REGION Network 3: Stopper02
   "InstSq_Stopper02"(INIT_SQ := #tempInit,   // "Sq_Process_Stopper"
                      ACK_EF := #tempAck,
                      SW_AUTO := #tempSwAuto,
                      SW_TAP := #tempSwTap,
                      SW_MAN := #tempSwMan,
                      T_PUSH := #tempPush,
                      ixStart := "InstSq_Process_Lift1".qxReadyForNextWT,
                      ixCarrierPresent := "FG_TS_Stopper02_B_Detect",
                      ixCheckTargetReached := true,
                      ixTargetReached := "FG_TS_Lift01_B_Detect",
                      itStopperRelease := t#150ms,
                      signals := #station.signals,
                      sq := #station.stepSeqs.stepSeq[2],
                      cylinder_stopper := "TransportActors".Stopper02);
END_REGION

REGION Network 4: Lift 1
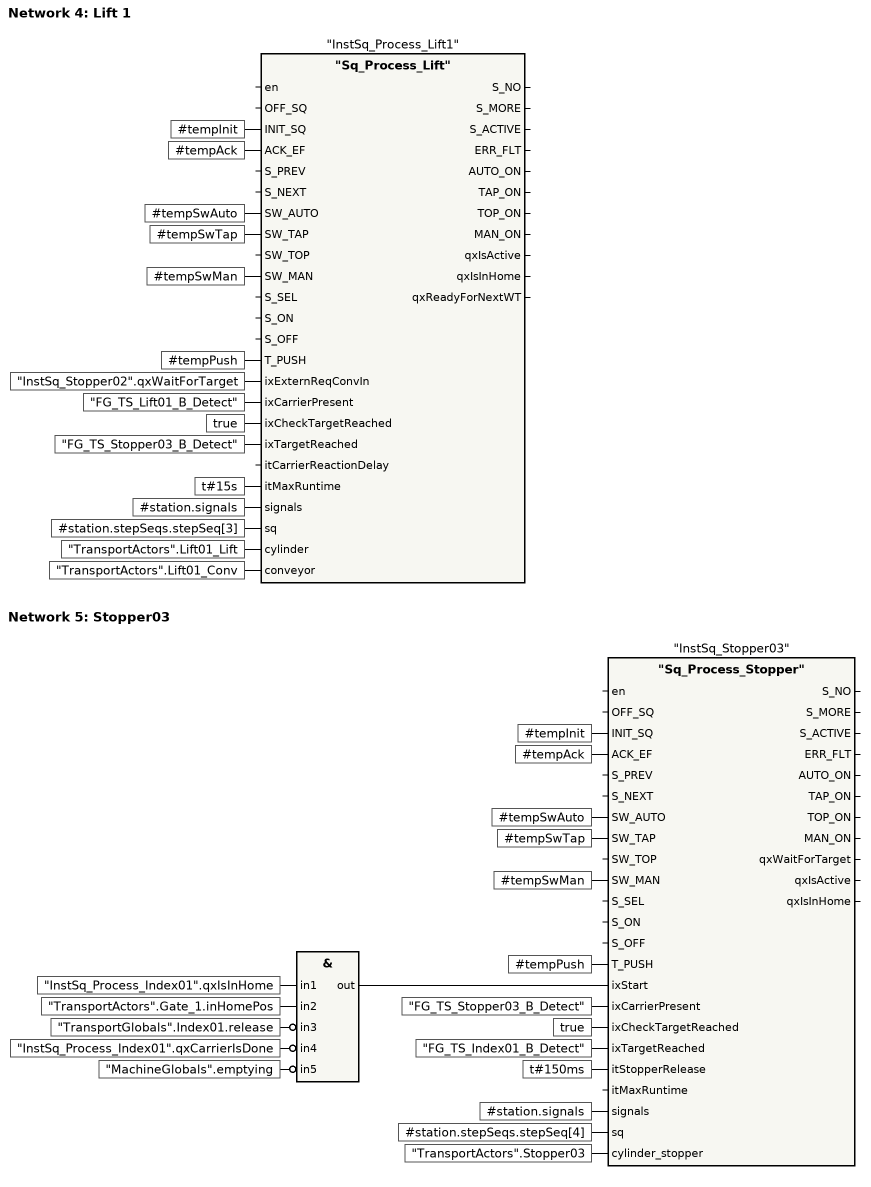
   "InstSq_Process_Lift1"(INIT_SQ := #tempInit,   // "Sq_Process_Lift"
                          ACK_EF := #tempAck,
                          SW_AUTO := #tempSwAuto,
                          SW_TAP := #tempSwTap,
                          SW_MAN := #tempSwMan,
                          T_PUSH := #tempPush,
                          ixExternReqConvIn := "InstSq_Stopper02".qxWaitForTarget,
                          ixCarrierPresent := "FG_TS_Lift01_B_Detect",
                          ixCheckTargetReached := true,
                          ixTargetReached := "FG_TS_Stopper03_B_Detect",
                          itMaxRuntime := t#15s,
                          signals := #station.signals,
                          sq := #station.stepSeqs.stepSeq[3],
                          cylinder := "TransportActors".Lift01_Lift,
                          conveyor := "TransportActors".Lift01_Conv);
END_REGION

REGION Network 5: Stopper03
   "InstSq_Stopper03"(INIT_SQ := #tempInit,   // "Sq_Process_Stopper"
                      ACK_EF := #tempAck,
                      SW_AUTO := #tempSwAuto,
                      SW_TAP := #tempSwTap,
                      SW_MAN := #tempSwMan,
                      T_PUSH := #tempPush,
                      ixStart := "InstSq_Process_Index01".qxIsInHome AND "TransportActors".Gate_1.inHomePos AND NOT "TransportGlobals".Index01.release AND NOT "InstSq_Process_Index01".qxCarrierIsDone AND NOT "MachineGlobals".emptying,
                      ixCarrierPresent := "FG_TS_Stopper03_B_Detect",
                      ixCheckTargetReached := true,
                      ixTargetReached := "FG_TS_Index01_B_Detect",
                      itStopperRelease := t#150ms,
                      signals := #station.signals,
                      sq := #station.stepSeqs.stepSeq[4],
                      cylinder_stopper := "TransportActors".Stopper03);
END_REGION

REGION Network 6: Index01
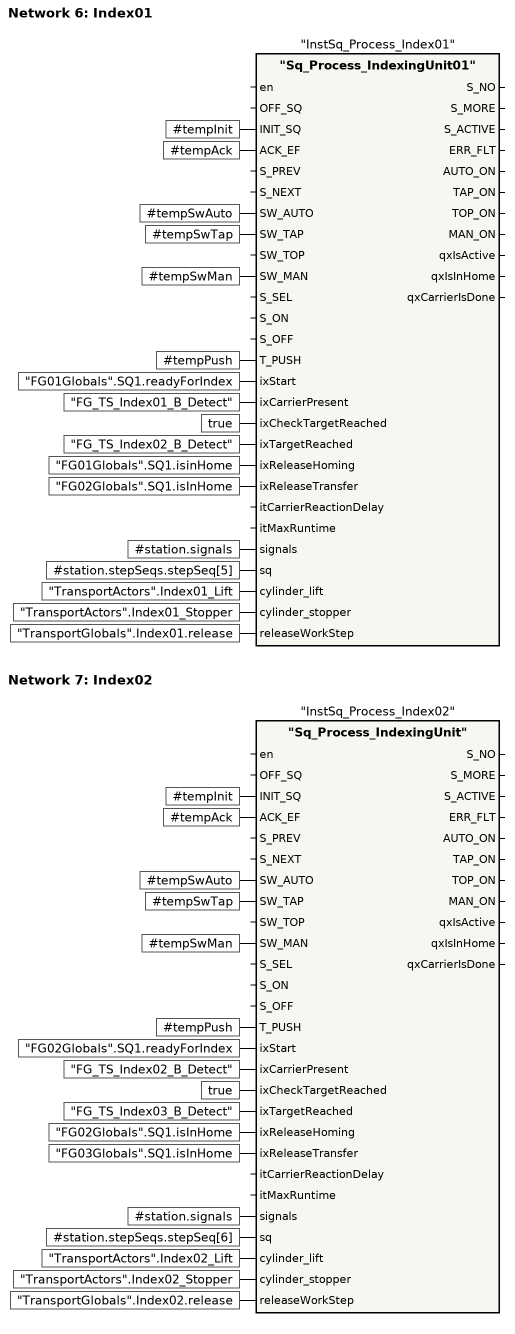
   "InstSq_Process_Index01"(INIT_SQ := #tempInit,   // "Sq_Process_IndexingUnit01"
                           ACK_EF := #tempAck,
                           SW_AUTO := #tempSwAuto,
                           SW_TAP := #tempSwTap,
                           SW_MAN := #tempSwMan,
                           T_PUSH := #tempPush,
                           ixStart := "FG01Globals".SQ1.readyForIndex,
                           ixCarrierPresent := "FG_TS_Index01_B_Detect",
                           ixCheckTargetReached := true,
                           ixTargetReached := "FG_TS_Index02_B_Detect",
                           ixReleaseHoming := "FG01Globals".SQ1.isinHome,
                           ixReleaseTransfer := "FG02Globals".SQ1.isInHome,
                           signals := #station.signals,
                           sq := #station.stepSeqs.stepSeq[5],
                           cylinder_lift := "TransportActors".Index01_Lift,
                           cylinder_stopper := "TransportActors".Index01_Stopper,
                           releaseWorkStep := "TransportGlobals".Index01.release);
END_REGION

REGION Network 7: Index02
   "InstSq_Process_Index02"(INIT_SQ := #tempInit,   // "Sq_Process_IndexingUnit"
                           ACK_EF := #tempAck,
                           SW_AUTO := #tempSwAuto,
                           SW_TAP := #tempSwTap,
                           SW_MAN := #tempSwMan,
                           T_PUSH := #tempPush,
                           ixStart := "FG02Globals".SQ1.readyForIndex,
                           ixCarrierPresent := "FG_TS_Index02_B_Detect",
                           ixCheckTargetReached := true,
                           ixTargetReached := "FG_TS_Index03_B_Detect",
                           ixReleaseHoming := "FG02Globals".SQ1.isInHome,
                           ixReleaseTransfer := "FG03Globals".SQ1.isInHome,
                           signals := #station.signals,
                           sq := #station.stepSeqs.stepSeq[6],
                           cylinder_lift := "TransportActors".Index02_Lift,
                           cylinder_stopper := "TransportActors".Index02_Stopper,
                           releaseWorkStep := "TransportGlobals".Index02.release);
END_REGION

REGION Network 8: Index03
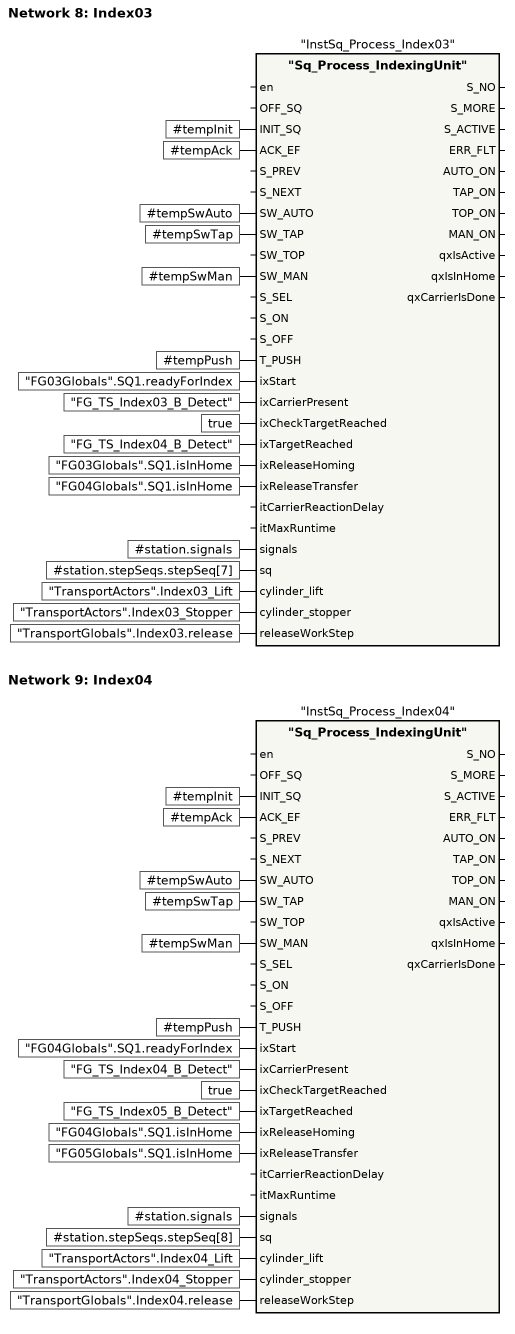
   "InstSq_Process_Index03"(INIT_SQ := #tempInit,   // "Sq_Process_IndexingUnit"
                           ACK_EF := #tempAck,
                           SW_AUTO := #tempSwAuto,
                           SW_TAP := #tempSwTap,
                           SW_MAN := #tempSwMan,
                           T_PUSH := #tempPush,
                           ixStart := "FG03Globals".SQ1.readyForIndex,
                           ixCarrierPresent := "FG_TS_Index03_B_Detect",
                           ixCheckTargetReached := true,
                           ixTargetReached := "FG_TS_Index04_B_Detect",
                           ixReleaseHoming := "FG03Globals".SQ1.isInHome,
                           ixReleaseTransfer := "FG04Globals".SQ1.isInHome,
                           signals := #station.signals,
                           sq := #station.stepSeqs.stepSeq[7],
                           cylinder_lift := "TransportActors".Index03_Lift,
                           cylinder_stopper := "TransportActors".Index03_Stopper,
                           releaseWorkStep := "TransportGlobals".Index03.release);
END_REGION

REGION Network 9: Index04
   "InstSq_Process_Index04"(INIT_SQ := #tempInit,   // "Sq_Process_IndexingUnit"
                           ACK_EF := #tempAck,
                           SW_AUTO := #tempSwAuto,
                           SW_TAP := #tempSwTap,
                           SW_MAN := #tempSwMan,
                           T_PUSH := #tempPush,
                           ixStart := "FG04Globals".SQ1.readyForIndex,
                           ixCarrierPresent := "FG_TS_Index04_B_Detect",
                           ixCheckTargetReached := true,
                           ixTargetReached := "FG_TS_Index05_B_Detect",
                           ixReleaseHoming := "FG04Globals".SQ1.isInHome,
                           ixReleaseTransfer := "FG05Globals".SQ1.isInHome,
                           signals := #station.signals,
                           sq := #station.stepSeqs.stepSeq[8],
                           cylinder_lift := "TransportActors".Index04_Lift,
                           cylinder_stopper := "TransportActors".Index04_Stopper,
                           releaseWorkStep := "TransportGlobals".Index04.release);
END_REGION

REGION Network 10: Index05
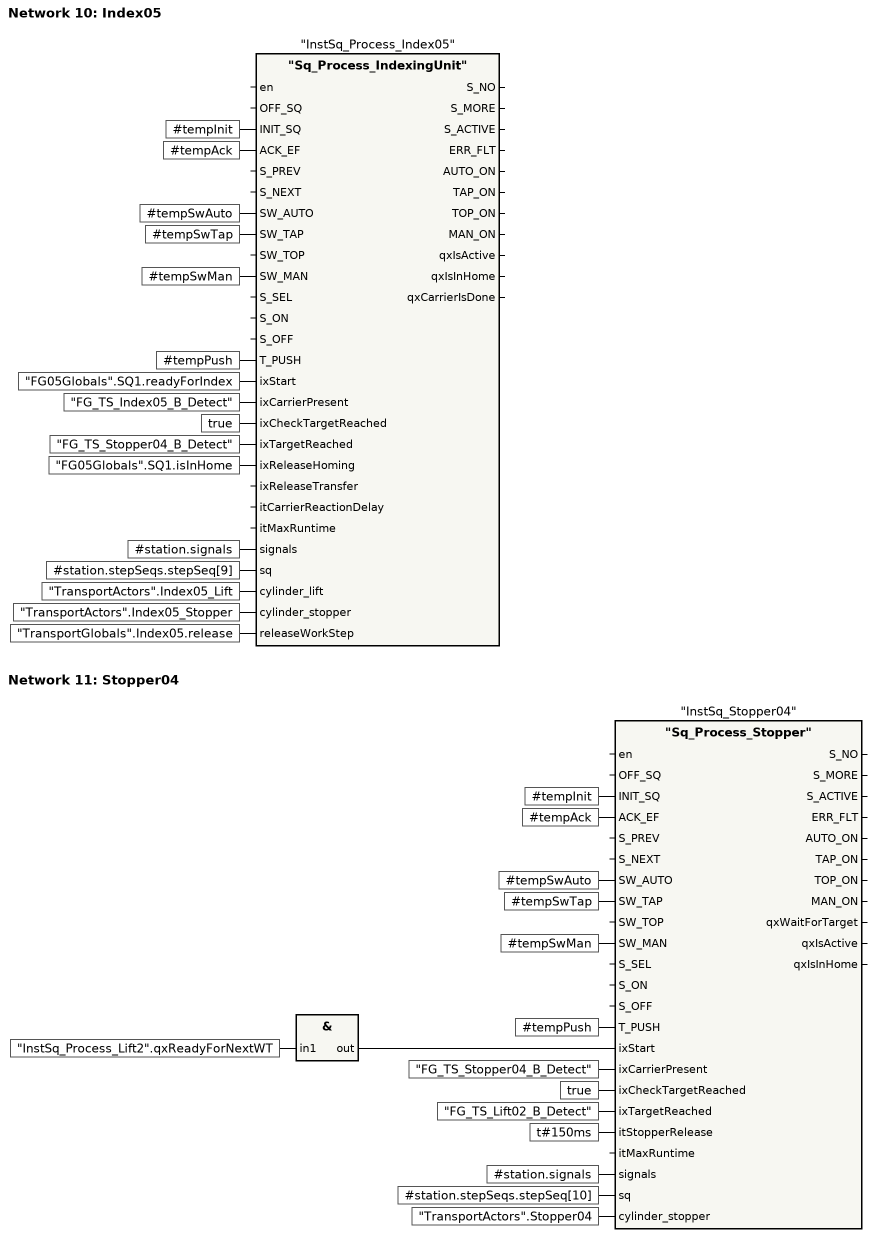
   "InstSq_Process_Index05"(INIT_SQ := #tempInit,   // "Sq_Process_IndexingUnit"
                           ACK_EF := #tempAck,
                           SW_AUTO := #tempSwAuto,
                           SW_TAP := #tempSwTap,
                           SW_MAN := #tempSwMan,
                           T_PUSH := #tempPush,
                           ixStart := "FG05Globals".SQ1.readyForIndex,
                           ixCarrierPresent := "FG_TS_Index05_B_Detect",
                           ixCheckTargetReached := true,
                           ixTargetReached := "FG_TS_Stopper04_B_Detect",
                           ixReleaseHoming := "FG05Globals".SQ1.isInHome,
                           signals := #station.signals,
                           sq := #station.stepSeqs.stepSeq[9],
                           cylinder_lift := "TransportActors".Index05_Lift,
                           cylinder_stopper := "TransportActors".Index05_Stopper,
                           releaseWorkStep := "TransportGlobals".Index05.release);
END_REGION

REGION Network 11: Stopper04
   "InstSq_Stopper04"(INIT_SQ := #tempInit,   // "Sq_Process_Stopper"
                      ACK_EF := #tempAck,
                      SW_AUTO := #tempSwAuto,
                      SW_TAP := #tempSwTap,
                      SW_MAN := #tempSwMan,
                      T_PUSH := #tempPush,
                      ixStart := "InstSq_Process_Lift2".qxReadyForNextWT,
                      ixCarrierPresent := "FG_TS_Stopper04_B_Detect",
                      ixCheckTargetReached := true,
                      ixTargetReached := "FG_TS_Lift02_B_Detect",
                      itStopperRelease := t#150ms,
                      signals := #station.signals,
                      sq := #station.stepSeqs.stepSeq[10],
                      cylinder_stopper := "TransportActors".Stopper04);
END_REGION

REGION Network 12: Lift 2
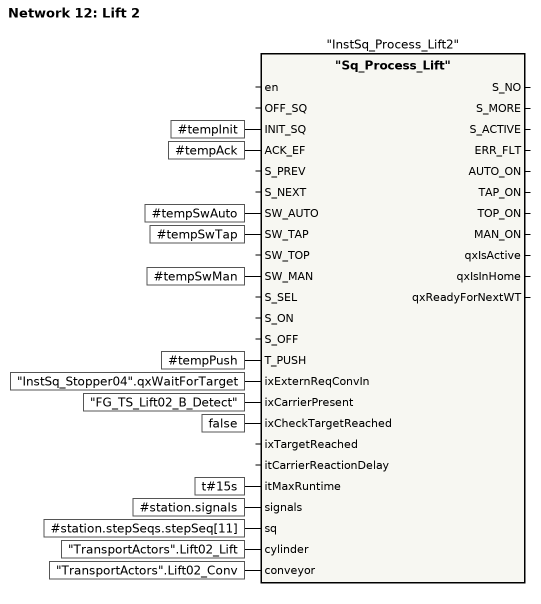
   "InstSq_Process_Lift2"(INIT_SQ := #tempInit,   // "Sq_Process_Lift"
                          ACK_EF := #tempAck,
                          SW_AUTO := #tempSwAuto,
                          SW_TAP := #tempSwTap,
                          SW_MAN := #tempSwMan,
                          T_PUSH := #tempPush,
                          ixExternReqConvIn := "InstSq_Stopper04".qxWaitForTarget,
                          ixCarrierPresent := "FG_TS_Lift02_B_Detect",
                          ixCheckTargetReached := false,
                          itMaxRuntime := t#15s,
                          signals := #station.signals,
                          sq := #station.stepSeqs.stepSeq[11],
                          cylinder := "TransportActors".Lift02_Lift,
                          conveyor := "TransportActors".Lift02_Conv);
END_REGION
END_FUNCTION

// folder: 9. Library

FUNCTION_BLOCK "MachineControl"   // FB9000, FBD
TITLE = Maschinensteuerung
{ S7_Optimized_Access := 'TRUE' }
VERSION : 0.1
// Ersteller: Andreas Fast Automation
// E-Mail: automation@fast-andreas.de
// 
// Projekt dient zu Demonstrationszwecken und frei genutzt werden.
// 
// Bausteinbeschreibung:
   VAR_INPUT
      firstPlcCycle : Bool;   // Erster Zyklus
      configNoControlOff : Bool := true;   // 1 = Ohne controlOff (Ein-/Ausschalten nur über controlOn)
      controlOn : Bool;   // Input 'control on' (if true)
      contolOff : Bool := true;   // Input 'control off' (if false)
      automaticMode : Bool;   // Input 'automatic/manual operation'
      singleStep : Bool;   // Input 'single step'
      autoStart : Bool;   // Input 'automatic start'
      autoStop : Bool;   // Input ' automatic stop'
      immediateStop : Bool;   // Input 'immediate stop'
      reset : Bool;   // Input 'machine reset'
      acknowledge : Bool;   // Input ' acknowledgement'
      errFlt : Bool;   // Input 'machine error'
   END_VAR
   VAR_OUTPUT
      controlOnLight : Bool;   // Steuerung Ein = Dauerlicht; Steuerung fährt hoch = Blinklicht; Steuerung aus = Licht aus
      setupOnLight : Bool;   // Einrichten aktiv = Ein
      automaticRunsLight : Bool;   // Automatik aktiv = Dauerlicht; Teilautomatik = Blinklicht; Automatik aus = Licht aus
      singleStepLight : Bool;   // Einzelschritt läuft = Dauerlicht
      automaticStopsLight : Bool;   // Automatik stoppt = Blinklicht
      errFltLight : Bool;   // Störung = Dauerlicht
      homingLight : Bool;   // Grundstellungsfahrt läuft = Blinklicht; Maschine in Grundstellung = Dauerlicht
      manAutoLight : Bool;   // Auto = Dauerlicht, Hand = Licht aus
   END_VAR
   VAR_IN_OUT
      safety : "typeMachineSafety";
      machine : "typeMachine";
      stations : "typeStations";
      manualMovement : "typeManualMovements";
      plcErrMsg : "typePlcErrMsg";
      hmiErrMsg : "typeHmiErrMsg";
   END_VAR
   VAR
      statControlRunUp : Bool;
      statTrigControlOn : Bool;
      statTrigReset : Bool;
      statTrigSingleStep : Bool;
      statTrigAutoStart : Bool;
      statTrigHomingDone : Bool;
      statFirstCycle : Bool;
      statStationsAllStopped : Bool;
      statStationsAllRunning : Bool;
      statAnyStationInAutoRun : Bool;
      instTonRunUp : TON_TIME;
      instAlarmHandler : "AlarmHandler";
   END_VAR
   VAR_TEMP
      tempStationError : Bool;
      tempStationsInSetup : Bool;
      tempAnyJogIsActive : Bool;
   END_VAR
   VAR_TEMP   // added for the SCL form of the ladder/FBD networks
      _w1 : Bool;
      _w2 : Bool;
   END_VAR
BEGIN

REGION Network 1: Meldungen auslösen
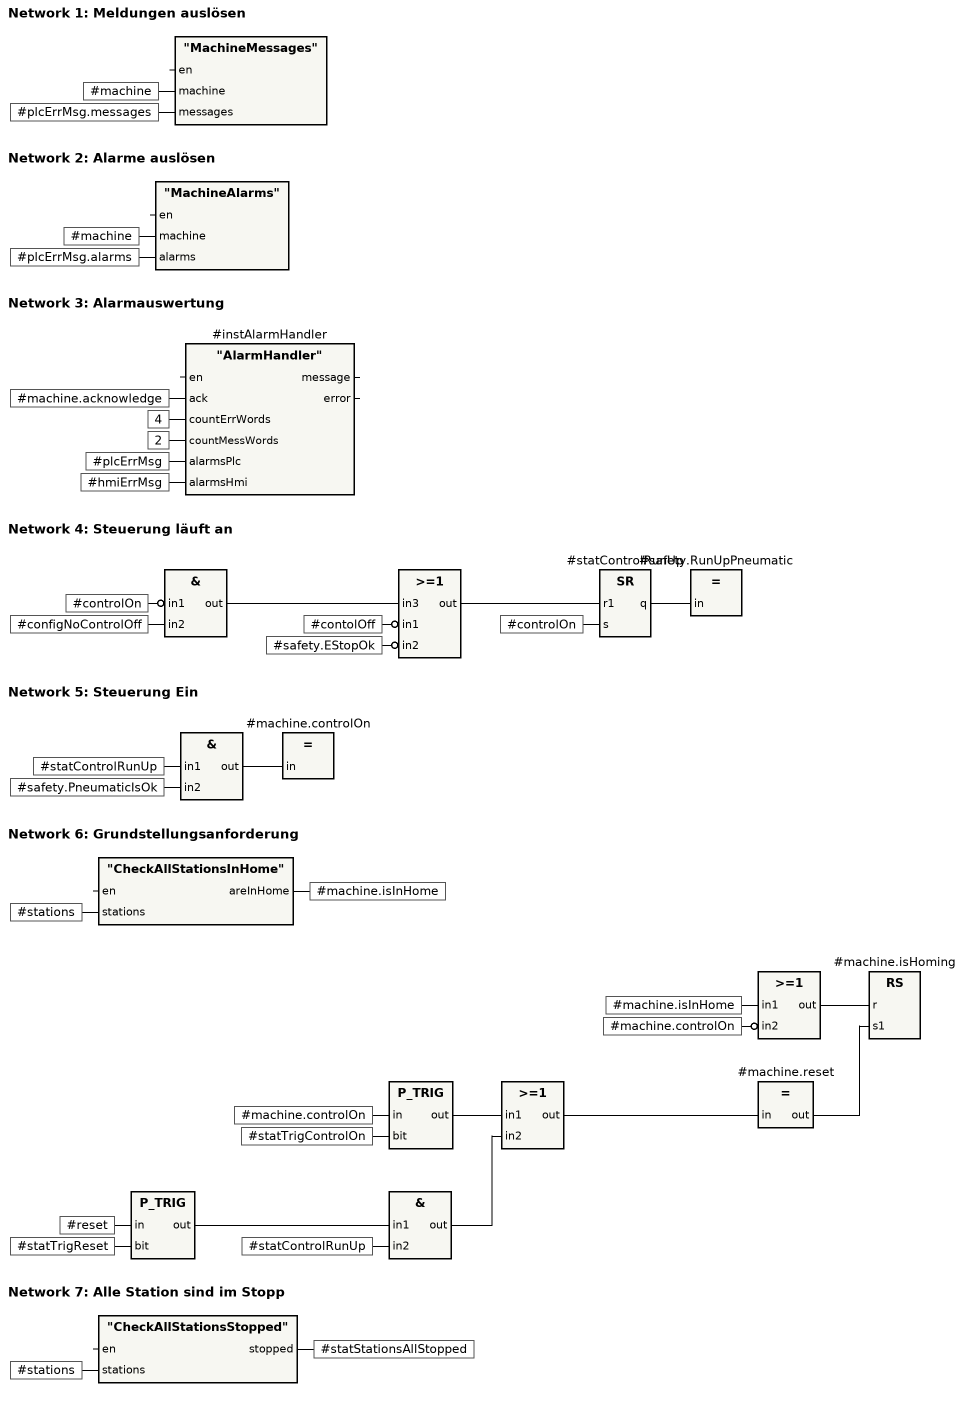
   "MachineMessages"(machine := #machine, messages := #plcErrMsg.messages);
END_REGION

REGION Network 2: Alarme auslösen
   "MachineAlarms"(machine := #machine, alarms := #plcErrMsg.alarms);
END_REGION

REGION Network 3: Alarmauswertung
   #instAlarmHandler(ack := #machine.acknowledge,   // "AlarmHandler"
                     countErrWords := 4,
                     countMessWords := 2,
                     alarmsPlc := #plcErrMsg,
                     alarmsHmi := #hmiErrMsg);
END_REGION

REGION Network 4: Steuerung läuft an
   IF #controlOn THEN
       #statControlRunUp := TRUE;   // SR flip-flop
   END_IF;
   IF (NOT #controlOn AND #configNoControlOff) OR NOT #contolOff OR NOT #safety.EStopOk THEN
       #statControlRunUp := FALSE;
   END_IF;
   #safety.RunUpPneumatic := #statControlRunUp;
END_REGION

REGION Network 5: Steuerung Ein
   #machine.controlOn := #statControlRunUp AND #safety.PneumaticIsOk;
END_REGION

REGION Network 6: Grundstellungsanforderung
   "CheckAllStationsInHome"(stations := #stations, areInHome => #machine.isInHome);
   #_w1 := #machine.controlOn AND NOT #statTrigControlOn;   // rising edge
   #statTrigControlOn := #machine.controlOn;
   #_w2 := #reset AND NOT #statTrigReset;   // rising edge
   #statTrigReset := #reset;
   #machine.reset := #_w1 OR (#_w2 AND #statControlRunUp);
   IF #machine.isInHome OR NOT #machine.controlOn THEN
       #machine.isHoming := FALSE;   // RS flip-flop
   END_IF;
   IF #machine.reset THEN #machine.isHoming := TRUE; END_IF;
END_REGION

REGION Network 7: Alle Station sind im Stopp
   "CheckAllStationsStopped"(stations := #stations, stopped => #statStationsAllStopped);
END_REGION

REGION Network 8: Automatikmodus
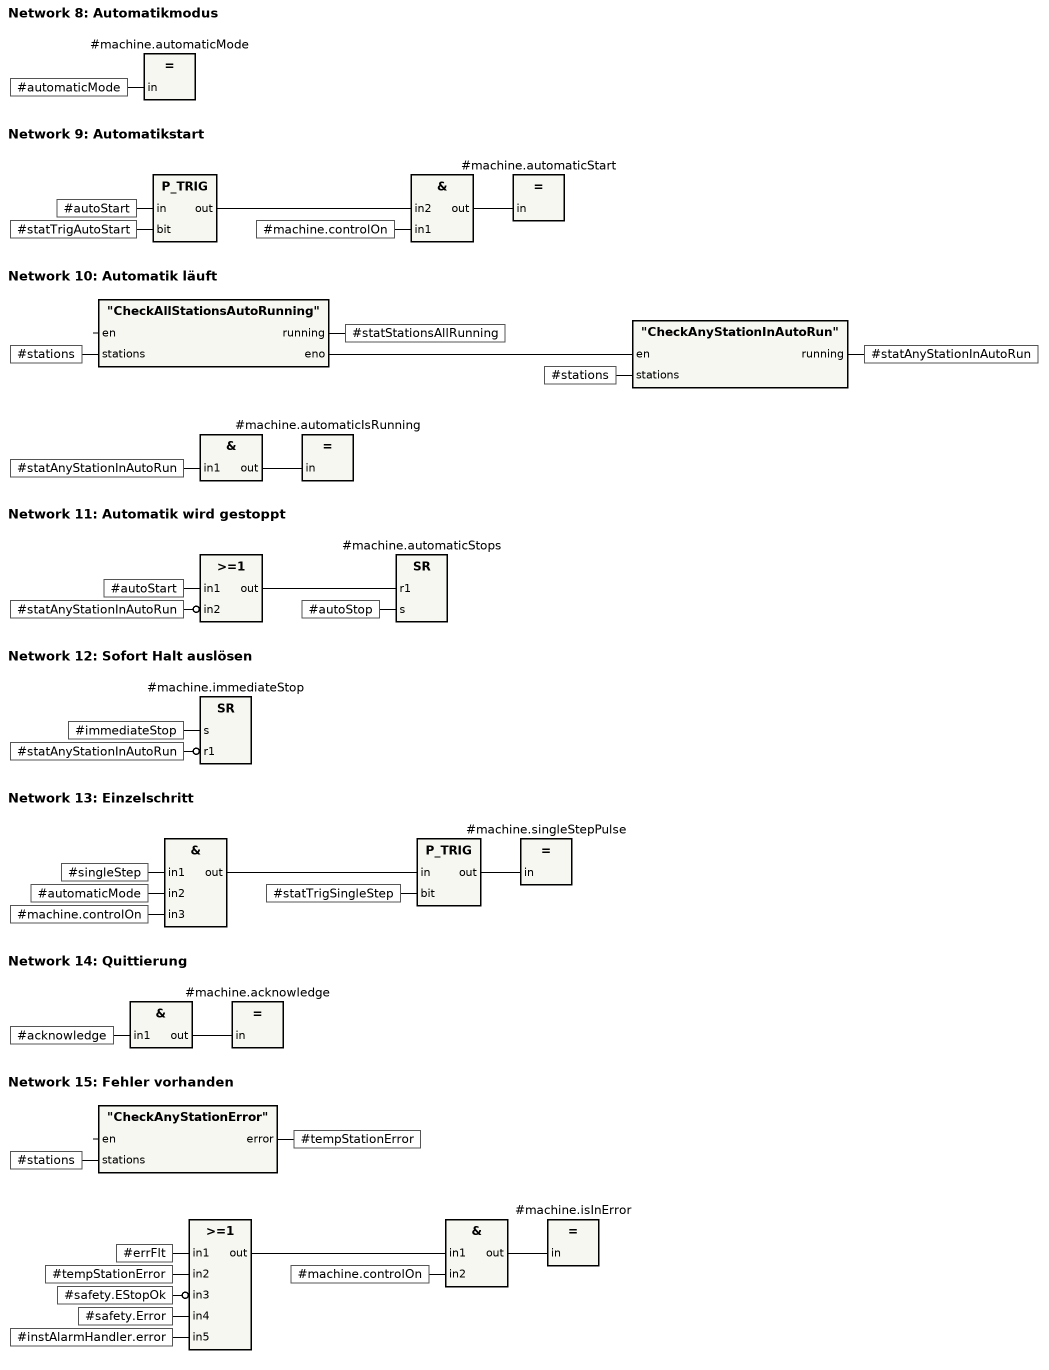
   #machine.automaticMode := #automaticMode;
END_REGION

REGION Network 9: Automatikstart
   #_w1 := #autoStart AND NOT #statTrigAutoStart;   // rising edge
   #statTrigAutoStart := #autoStart;
   #machine.automaticStart := #_w1 AND #machine.controlOn;
END_REGION

REGION Network 10: Automatik läuft
   "CheckAllStationsAutoRunning"(stations := #stations, running => #statStationsAllRunning, ENO => #_w1);
   IF #_w1 THEN
       "CheckAnyStationInAutoRun"(stations := #stations, running => #statAnyStationInAutoRun);
   END_IF;
   #machine.automaticIsRunning := #statAnyStationInAutoRun;
END_REGION

REGION Network 11: Automatik wird gestoppt
   IF #autoStop THEN
       #machine.automaticStops := TRUE;   // SR flip-flop
   END_IF;
   IF #autoStart OR NOT #statAnyStationInAutoRun THEN #machine.automaticStops := FALSE; END_IF;
END_REGION

REGION Network 12: Sofort Halt auslösen
   IF #immediateStop THEN
       #machine.immediateStop := TRUE;   // SR flip-flop
   END_IF;
   IF NOT #statAnyStationInAutoRun THEN #machine.immediateStop := FALSE; END_IF;
END_REGION

REGION Network 13: Einzelschritt
   #_w1 := #singleStep AND #automaticMode AND #machine.controlOn;
   #_w2 := #_w1 AND NOT #statTrigSingleStep;   // rising edge
   #statTrigSingleStep := #_w1;
   #machine.singleStepPulse := #_w2;
END_REGION

REGION Network 14: Quittierung
   #machine.acknowledge := #acknowledge;
END_REGION

REGION Network 15: Fehler vorhanden
   "CheckAnyStationError"(stations := #stations, error => #tempStationError);
   #machine.isInError := (#errFlt OR #tempStationError OR NOT #safety.EStopOk OR #safety.Error OR #instAlarmHandler.error) AND #machine.controlOn;
END_REGION

REGION Network 16: Initialisierung Bewegungsfunktionen (Teil 1)
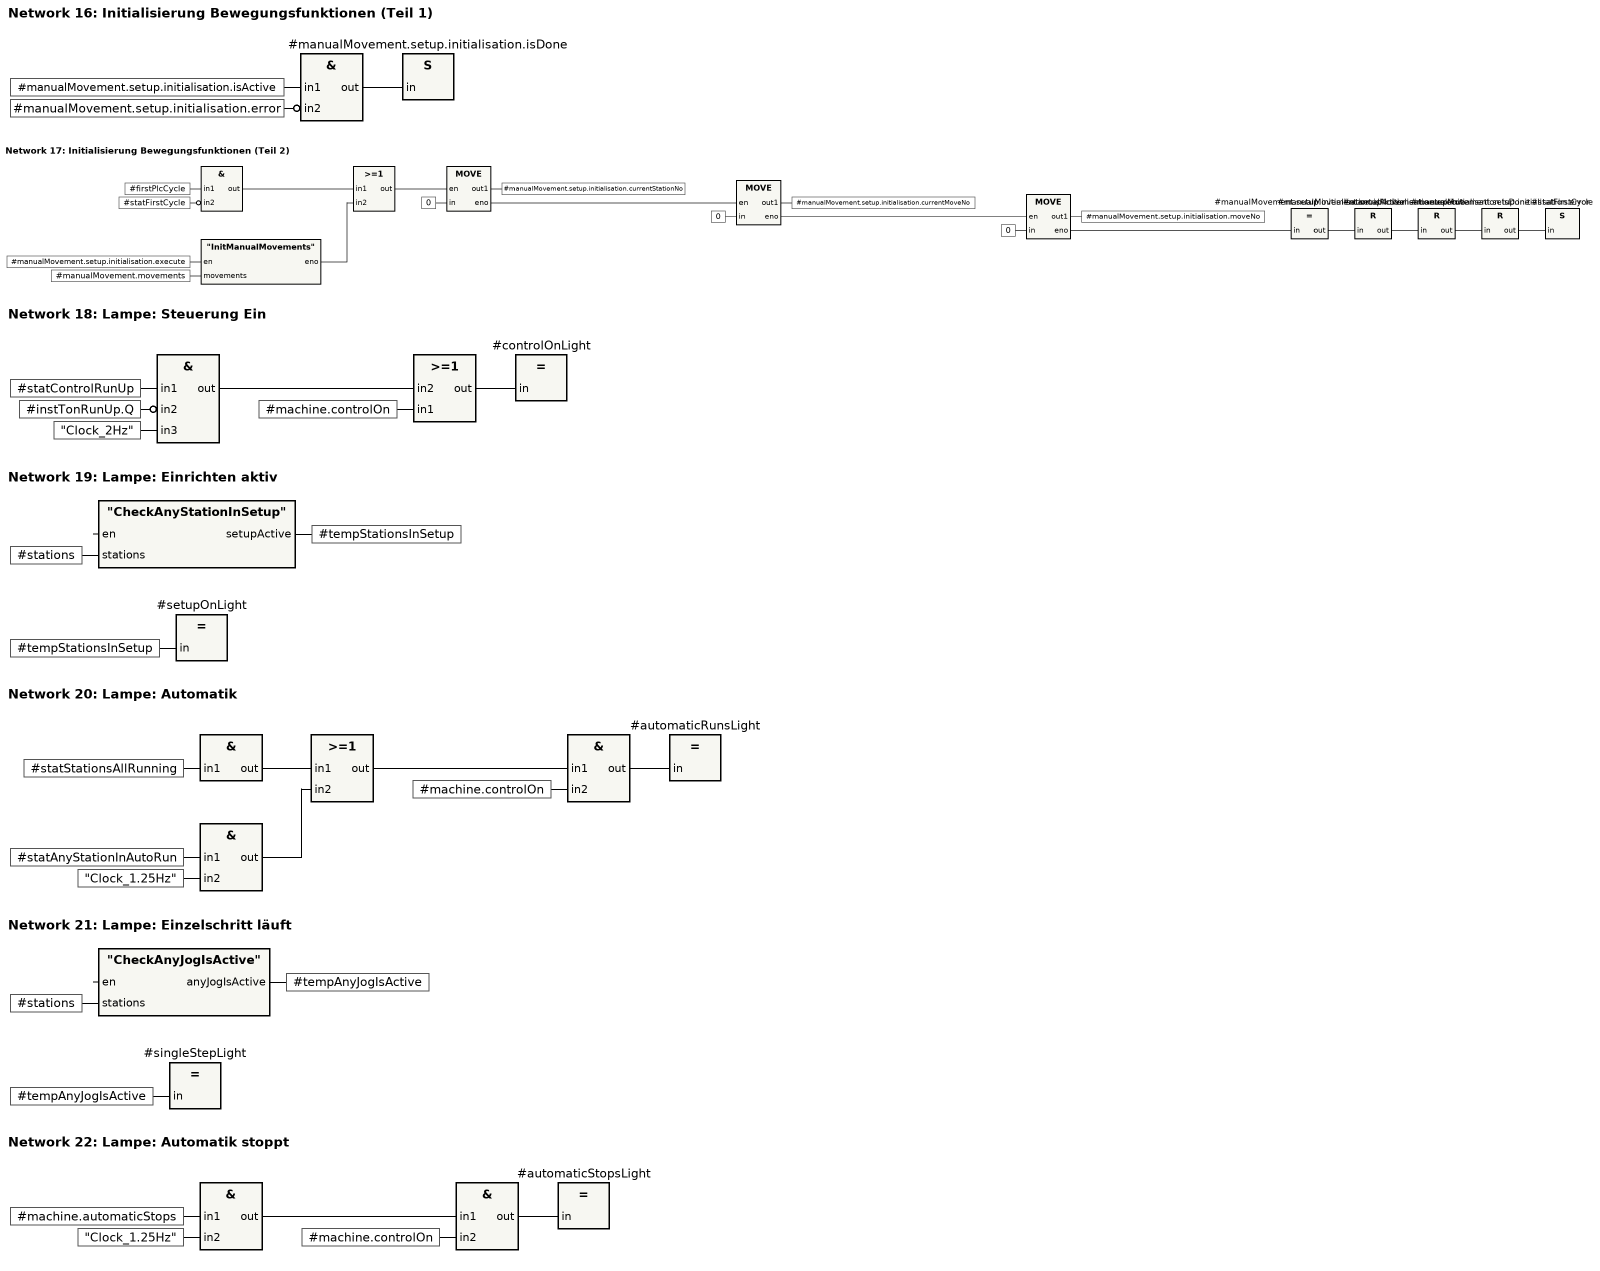
   IF #manualMovement.setup.initialisation.isActive AND NOT #manualMovement.setup.initialisation.error THEN
       #manualMovement.setup.initialisation.isDone := TRUE;
   END_IF;
END_REGION

REGION Network 17: Initialisierung Bewegungsfunktionen (Teil 2)
   "InitManualMovements"(EN := #manualMovement.setup.initialisation.execute,
                         movements := #manualMovement.movements,
                         ENO => #_w1);
   #_w2 := (#firstPlcCycle AND NOT #statFirstCycle) OR #_w1;
   IF #_w2 THEN
       #manualMovement.setup.initialisation.currentStationNo := 0;
       #manualMovement.setup.initialisation.currentMoveNo := 0;
       #manualMovement.setup.initialisation.moveNo := 0;
   END_IF;
   #manualMovement.setup.initialisation.isActive := #_w2;
   IF #_w2 THEN
       #manualMovement.setup.initialisation.execute := FALSE;
       #manualMovement.setup.initialisation.isDone := FALSE;
       #manualMovement.setup.initialisation.error := FALSE;
       #statFirstCycle := TRUE;
   END_IF;
END_REGION

REGION Network 18: Lampe: Steuerung Ein
   #controlOnLight := (#statControlRunUp AND NOT #instTonRunUp.Q AND "Clock_2Hz") OR #machine.controlOn;
END_REGION

REGION Network 19: Lampe: Einrichten aktiv
   "CheckAnyStationInSetup"(stations := #stations, setupActive => #tempStationsInSetup);
   #setupOnLight := #tempStationsInSetup;
END_REGION

REGION Network 20: Lampe: Automatik
   #automaticRunsLight := (#statStationsAllRunning OR (#statAnyStationInAutoRun AND "Clock_1.25Hz")) AND #machine.controlOn;
END_REGION

REGION Network 21: Lampe: Einzelschritt läuft
   "CheckAnyJogIsActive"(stations := #stations, anyJogIsActive => #tempAnyJogIsActive);
   #singleStepLight := #tempAnyJogIsActive;
END_REGION

REGION Network 22: Lampe: Automatik stoppt
   #automaticStopsLight := #machine.automaticStops AND "Clock_1.25Hz" AND #machine.controlOn;
END_REGION

REGION Network 23: Lampe: Fehler
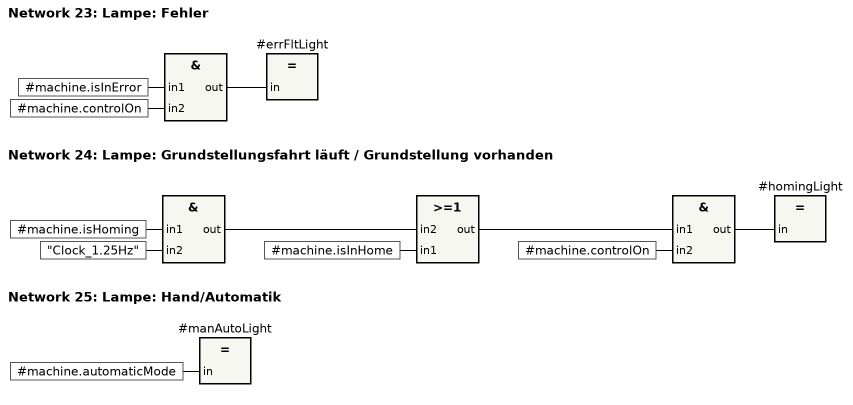
   #errFltLight := #machine.isInError AND #machine.controlOn;
END_REGION

REGION Network 24: Lampe: Grundstellungsfahrt läuft / Grundstellung vorhanden
   #homingLight := ((#machine.isHoming AND "Clock_1.25Hz") OR #machine.isInHome) AND #machine.controlOn;
END_REGION

REGION Network 25: Lampe: Hand/Automatik
   #manAutoLight := #machine.automaticMode;
END_REGION
END_FUNCTION_BLOCK

FUNCTION_BLOCK "StationControl"   // FB9001, FBD
TITLE = Steuerung Station
{ S7_Optimized_Access := 'TRUE' }
VERSION : 0.1
// Ersteller: Andreas Fast Automation
// E-Mail: automation@fast-andreas.de
// 
// Projekt dient zu Demonstrationszwecken und frei genutzt werden.
// 
// Bausteinbeschreibung:
   VAR_INPUT
      stationNo : Int := 1;   // Stationsnummer
      safetyOk : Bool;   // Schutzkreis geschlossen
      autoStart : Bool;   // Automatikstart
      autoStop : Bool;   // Automatikstopp
      singlePulse : Bool;   // Einzelschritt (Halbautomatik)
      reset : Bool;   // Station rücksetzen/Grundstellungsfahrt starten
      ack : Bool;   // Quittieren
      error : Bool;   // Störung vorhanden
      robotsStopped : Bool := true;   // Roboter sind angehalten
   END_VAR
   VAR_IN_OUT
      exists : Bool;   // Station existiert
      machine : "typeMachine";
      station : "typeStationSignals";
      stepSeqs : "typeStepSequences";
      setup : "typeManualMoveSetup";
      plcErrMsg : "typePlcErrMsg";
      hmiErrMsg : "typeHmiErrMsg";
   END_VAR
   VAR
      statTrigReset : Bool;
      statTrigSinglePulse : Bool;
      statTrigHomingDone : Bool;
      sxTrigAutomaticMode : Bool;
      sxTrigTap : Bool;
      sxTrigAuto : Bool;
      instAlarmHandler : "AlarmHandler";
      tonTEST : TON_TIME;
   END_VAR
   VAR_TEMP
      tempHomingDone : Bool;
      tempSqInError : Bool;
      tempSqAllInHome : Bool;
      tempSqAllJogDone : Bool;
      tempSqsAreWaitingOrInError : Bool;
      tempSinglePulse : Bool;
   END_VAR
   VAR_TEMP   // added for the SCL form of the ladder/FBD networks
      _w1 : Bool;
      _w2 : Bool;
      _w3 : Bool;
   END_VAR
BEGIN

REGION Network 1: Station ist vorhanden / nicht reserviert
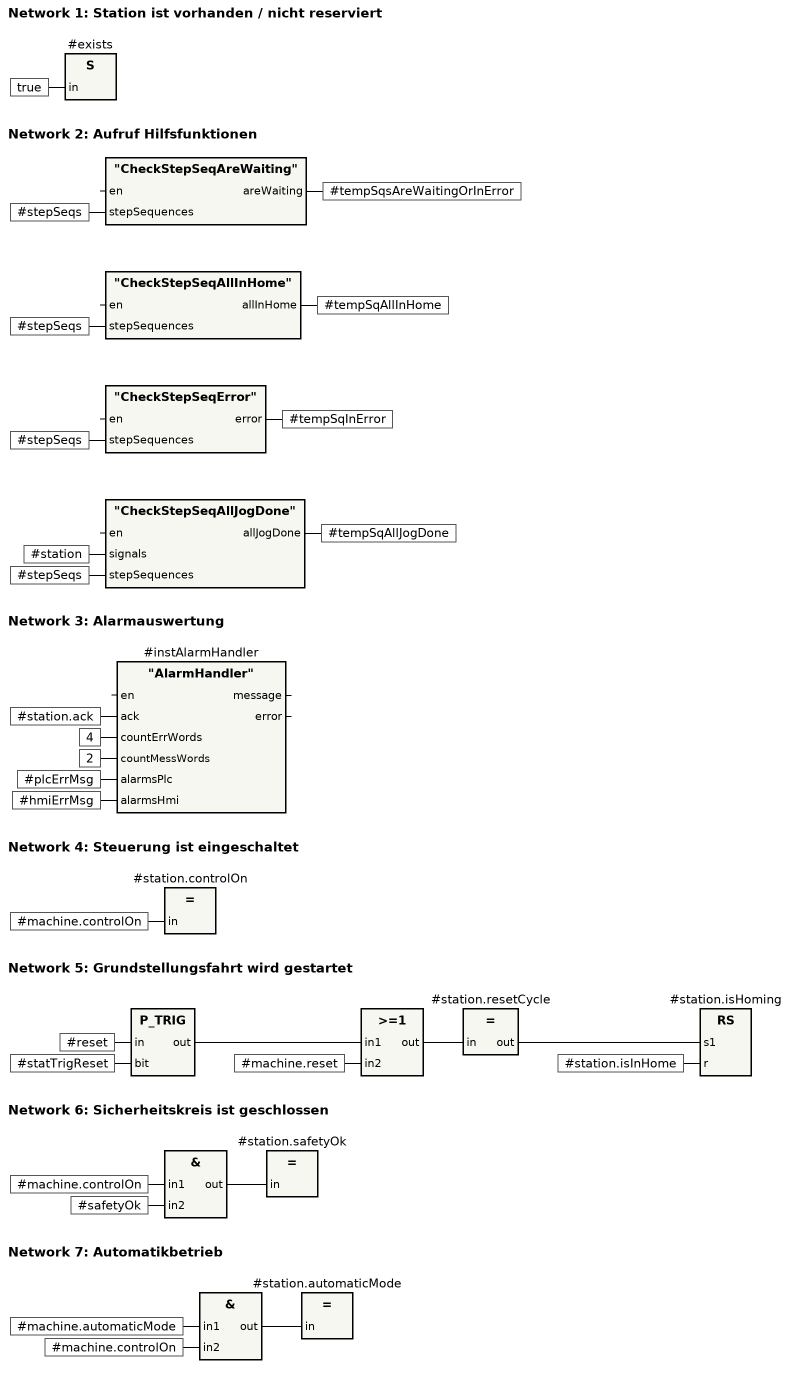
   IF true THEN #exists := TRUE; END_IF;
END_REGION

REGION Network 2: Aufruf Hilfsfunktionen
   "CheckStepSeqAreWaiting"(stepSequences := #stepSeqs, areWaiting => #tempSqsAreWaitingOrInError);
   "CheckStepSeqAllInHome"(stepSequences := #stepSeqs, allInHome => #tempSqAllInHome);
   "CheckStepSeqError"(stepSequences := #stepSeqs, error => #tempSqInError);
   "CheckStepSeqAllJogDone"(signals := #station, stepSequences := #stepSeqs, allJogDone => #tempSqAllJogDone);
END_REGION

REGION Network 3: Alarmauswertung
   #instAlarmHandler(ack := #station.ack,   // "AlarmHandler"
                     countErrWords := 4,
                     countMessWords := 2,
                     alarmsPlc := #plcErrMsg,
                     alarmsHmi := #hmiErrMsg);
END_REGION

REGION Network 4: Steuerung ist eingeschaltet
   #station.controlOn := #machine.controlOn;
END_REGION

REGION Network 5: Grundstellungsfahrt wird gestartet
   #_w1 := #reset AND NOT #statTrigReset;   // rising edge
   #statTrigReset := #reset;
   #station.resetCycle := #_w1 OR #machine.reset;
   IF #station.isInHome THEN
       #station.isHoming := FALSE;   // RS flip-flop
   END_IF;
   IF #station.resetCycle THEN #station.isHoming := TRUE; END_IF;
END_REGION

REGION Network 6: Sicherheitskreis ist geschlossen
   #station.safetyOk := #machine.controlOn AND #safetyOk;
END_REGION

REGION Network 7: Automatikbetrieb
   #station.automaticMode := #machine.automaticMode AND #machine.controlOn;
END_REGION

REGION Network 8: Handbetrieb
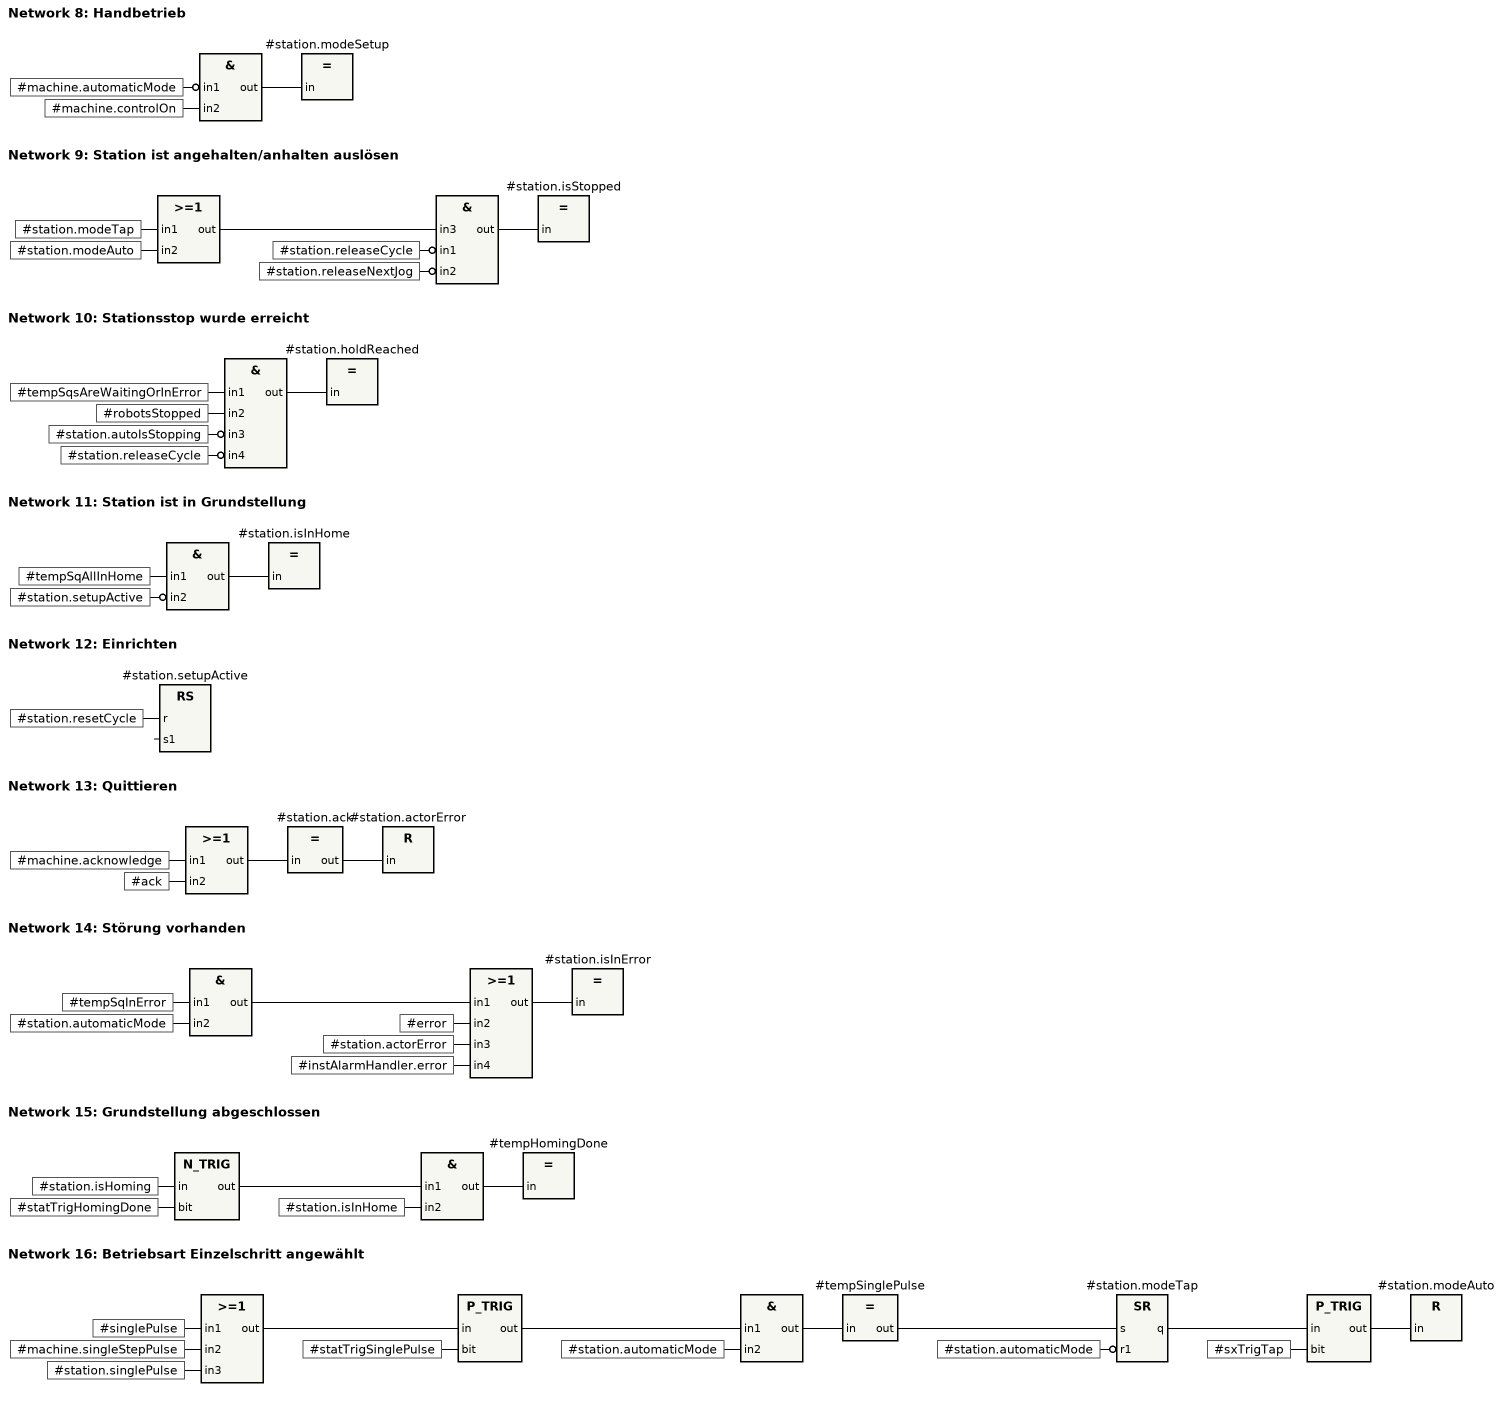
   #station.modeSetup := NOT #machine.automaticMode AND #machine.controlOn;
END_REGION

REGION Network 9: Station ist angehalten/anhalten auslösen
   #station.isStopped := (#station.modeTap OR #station.modeAuto) AND NOT #station.releaseCycle AND NOT #station.releaseNextJog;
END_REGION

REGION Network 10: Stationsstop wurde erreicht
   #station.holdReached := #tempSqsAreWaitingOrInError AND #robotsStopped AND NOT #station.autoIsStopping AND NOT #station.releaseCycle;
END_REGION

REGION Network 11: Station ist in Grundstellung
   #station.isInHome := #tempSqAllInHome AND NOT #station.setupActive;
END_REGION

REGION Network 12: Einrichten
   IF #station.resetCycle THEN
       #station.setupActive := FALSE;   // RS flip-flop
   END_IF;
END_REGION

REGION Network 13: Quittieren
   #station.ack := #machine.acknowledge OR #ack;
   IF #station.ack THEN #station.actorError := FALSE; END_IF;
END_REGION

REGION Network 14: Störung vorhanden
   #station.isInError := (#tempSqInError AND #station.automaticMode) OR #error OR #station.actorError OR #instAlarmHandler.error;
END_REGION

REGION Network 15: Grundstellung abgeschlossen
   #_w1 := NOT #station.isHoming AND #statTrigHomingDone;   // falling edge
   #statTrigHomingDone := #station.isHoming;
   #tempHomingDone := #_w1 AND #station.isInHome;
END_REGION

REGION Network 16: Betriebsart Einzelschritt angewählt
   #_w1 := #singlePulse OR #machine.singleStepPulse OR #station.singlePulse;
   #_w2 := #_w1 AND NOT #statTrigSinglePulse;   // rising edge
   #statTrigSinglePulse := #_w1;
   #tempSinglePulse := #_w2 AND #station.automaticMode;
   IF #tempSinglePulse THEN
       #station.modeTap := TRUE;   // SR flip-flop
   END_IF;
   IF NOT #station.automaticMode THEN #station.modeTap := FALSE; END_IF;
   #_w3 := #station.modeTap AND NOT #sxTrigTap;   // rising edge
   #sxTrigTap := #station.modeTap;
   IF #_w3 THEN #station.modeAuto := FALSE; END_IF;
END_REGION

REGION Network 17: Betriebsart Automatikbetrieb angewählt
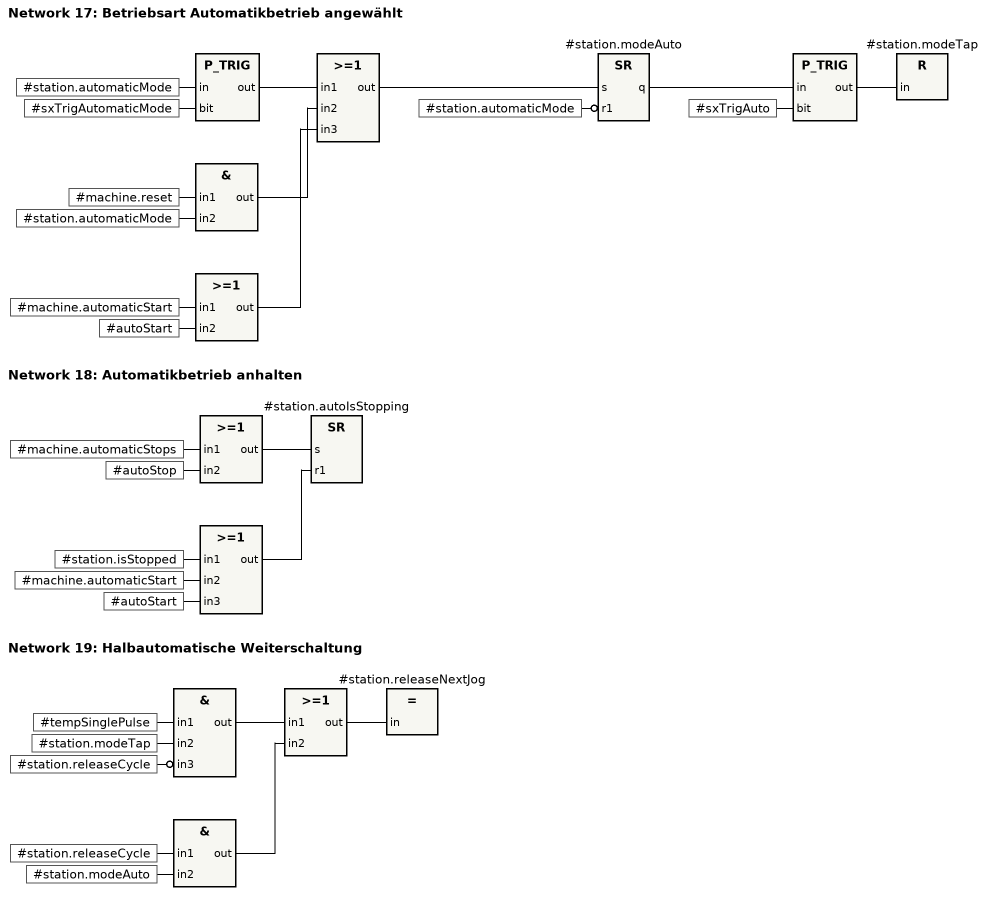
   #_w1 := #station.automaticMode AND NOT #sxTrigAutomaticMode;   // rising edge
   #sxTrigAutomaticMode := #station.automaticMode;
   IF #_w1 OR (#machine.reset AND #station.automaticMode) OR #machine.automaticStart OR #autoStart THEN
       #station.modeAuto := TRUE;   // SR flip-flop
   END_IF;
   IF NOT #station.automaticMode THEN #station.modeAuto := FALSE; END_IF;
   #_w2 := #station.modeAuto AND NOT #sxTrigAuto;   // rising edge
   #sxTrigAuto := #station.modeAuto;
   IF #_w2 THEN #station.modeTap := FALSE; END_IF;
END_REGION

REGION Network 18: Automatikbetrieb anhalten
   IF #machine.automaticStops OR #autoStop THEN
       #station.autoIsStopping := TRUE;   // SR flip-flop
   END_IF;
   IF #station.isStopped OR #machine.automaticStart OR #autoStart THEN
       #station.autoIsStopping := FALSE;
   END_IF;
END_REGION

REGION Network 19: Halbautomatische Weiterschaltung
   #station.releaseNextJog := (#tempSinglePulse AND #station.modeTap AND NOT #station.releaseCycle) OR (#station.releaseCycle AND #station.modeAuto);
END_REGION

REGION Network 20: Bearbeitungsfreigabe
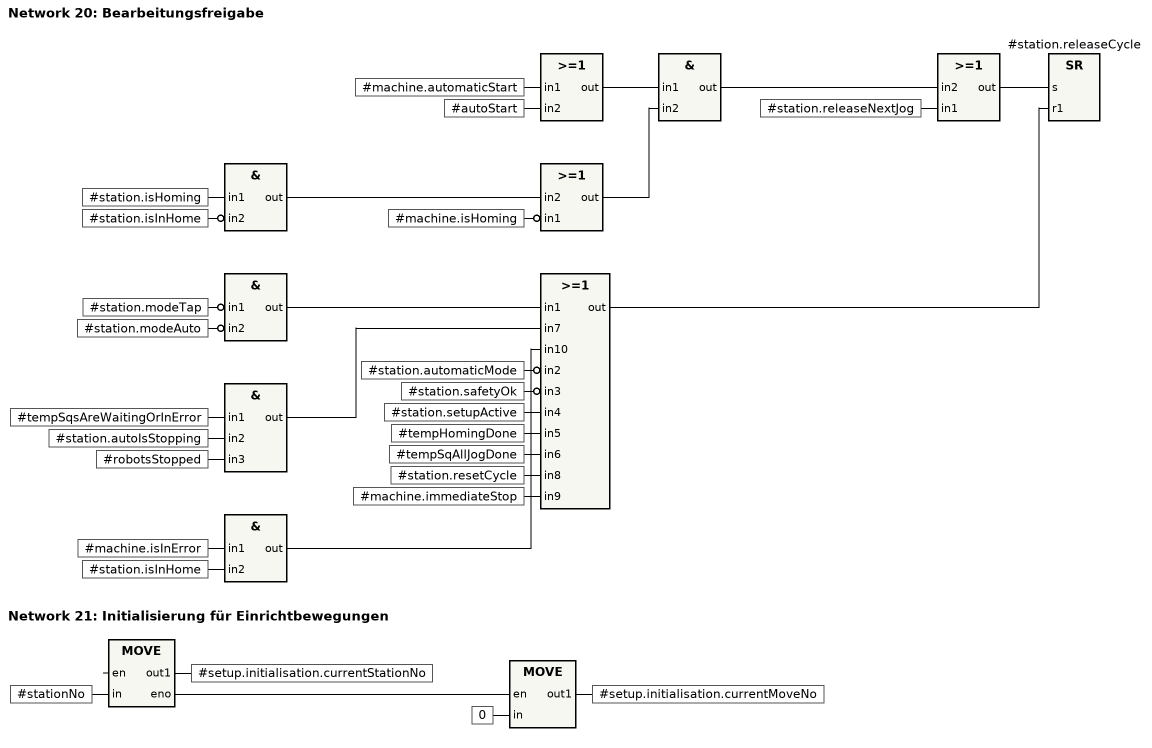
   IF ((#machine.automaticStart OR #autoStart) AND ((#station.isHoming AND NOT #station.isInHome) OR NOT #machine.isHoming)) OR #station.releaseNextJog THEN
       #station.releaseCycle := TRUE;   // SR flip-flop
   END_IF;
   IF (NOT #station.modeTap AND NOT #station.modeAuto) OR (#tempSqsAreWaitingOrInError AND #station.autoIsStopping AND #robotsStopped) OR (#machine.isInError AND #station.isInHome) OR NOT #station.automaticMode OR NOT #station.safetyOk OR #station.setupActive OR #tempHomingDone OR #tempSqAllJogDone OR #station.resetCycle OR #machine.immediateStop THEN
       #station.releaseCycle := FALSE;
   END_IF;
END_REGION

REGION Network 21: Initialisierung für Einrichtbewegungen
   #setup.initialisation.currentStationNo := #stationNo;
   #setup.initialisation.currentMoveNo := 0;
END_REGION
END_FUNCTION_BLOCK

FUNCTION_BLOCK "AlarmHandler"   // FB9009, SCL
{ S7_Optimized_Access := 'TRUE' }
VERSION : 0.1
   VAR_INPUT
      ack : Bool;   // Quittierung
      countErrWords : Int := 4;   // Anzahl Fehlermelde-Wörter
      countMessWords : Int;
   END_VAR
   VAR_OUTPUT
      message : Bool;
      error : Bool;   // Mindestens ein Fehler steht an
   END_VAR
   VAR_IN_OUT
      alarmsPlc : "typePlcErrMsg";
      alarmsHmi : "typeHmiErrMsg";
   END_VAR
   VAR
      risAck : Bool;
      instRisTrigger : R_TRIG;
      instTpAck : TP_TIME;
   END_VAR
   VAR_TEMP
      ackPulse : Bool;
      i : Int;
      x : Int;
      lengthPlcErrors : Int;
      lengthPlcMessages : Int;
   END_VAR
BEGIN
   // Ersteller: Andreas Fast Automation
   // E-Mail: automation@fast-andreas.de
   //
   // Projekt dient zu Demonstrationszwecken und frei genutzt werden.
   //
   // Bausteinbeschreibung:
   // 

   // Init values
   #lengthPlcErrors := #countErrWords * 16;
   #lengthPlcMessages := #countMessWords * 16;

   #instRisTrigger(CLK := #ack,
                   Q => #risAck);


   #instTpAck(IN:=#risAck,
              PT:=t#1s,
              Q=>#ackPulse);

   // Acknowledge signals for HMI
   FOR #i := 1 TO #countErrWords DO
       IF #ackPulse THEN
           #alarmsHmi.alarmAckPlc[#i + #countErrWords] := 16#FFFF;
       ELSE
           #alarmsHmi.alarmAckPlc[#i + #countErrWords] := 16#0;
       END_IF;
   END_FOR;


   // Clear errors of PLC
   IF #risAck THEN
       FOR #i := 1 TO #lengthPlcErrors DO
           #alarmsPlc.alarms.errorNo[#i] := FALSE;
       END_FOR;
   END_IF;

   // Assign plc alarms to HMI triggers
   FOR #i := 1 TO #countErrWords DO
       #x := (#i - 1) * 16;

       #alarmsHmi.alarmAckPlc[#i].%X0 := #alarmsPlc.alarms.errorNo[#x + 1];
       #alarmsHmi.alarmAckPlc[#i].%X1 := #alarmsPlc.alarms.errorNo[#x + 2];
       #alarmsHmi.alarmAckPlc[#i].%X2 := #alarmsPlc.alarms.errorNo[#x + 3];
       #alarmsHmi.alarmAckPlc[#i].%X3 := #alarmsPlc.alarms.errorNo[#x + 4];
       #alarmsHmi.alarmAckPlc[#i].%X4 := #alarmsPlc.alarms.errorNo[#x + 5];
       #alarmsHmi.alarmAckPlc[#i].%X5 := #alarmsPlc.alarms.errorNo[#x + 6];
       #alarmsHmi.alarmAckPlc[#i].%X6 := #alarmsPlc.alarms.errorNo[#x + 7];
       #alarmsHmi.alarmAckPlc[#i].%X7 := #alarmsPlc.alarms.errorNo[#x + 8];
       #alarmsHmi.alarmAckPlc[#i].%X8 := #alarmsPlc.alarms.errorNo[#x + 9];
       #alarmsHmi.alarmAckPlc[#i].%X9 := #alarmsPlc.alarms.errorNo[#x + 10];
       #alarmsHmi.alarmAckPlc[#i].%X10 := #alarmsPlc.alarms.errorNo[#x + 11];
       #alarmsHmi.alarmAckPlc[#i].%X11 := #alarmsPlc.alarms.errorNo[#x + 12];
       #alarmsHmi.alarmAckPlc[#i].%X12 := #alarmsPlc.alarms.errorNo[#x + 13];
       #alarmsHmi.alarmAckPlc[#i].%X13 := #alarmsPlc.alarms.errorNo[#x + 14];
       #alarmsHmi.alarmAckPlc[#i].%X14 := #alarmsPlc.alarms.errorNo[#x + 15];
       #alarmsHmi.alarmAckPlc[#i].%X15 := #alarmsPlc.alarms.errorNo[#x + 16];
   END_FOR;

   // Assign PLC messages to HMI messages
   FOR #i := 1 TO #countMessWords DO
       #x := (#i - 1) * 16;

       #alarmsHmi.message[#i].%X0 := #alarmsPlc.messages.msgNo[#x + 1];
       #alarmsHmi.message[#i].%X1 := #alarmsPlc.messages.msgNo[#x + 2];
       #alarmsHmi.message[#i].%X2 := #alarmsPlc.messages.msgNo[#x + 3];
       #alarmsHmi.message[#i].%X3 := #alarmsPlc.messages.msgNo[#x + 4];
       #alarmsHmi.message[#i].%X4 := #alarmsPlc.messages.msgNo[#x + 5];
       #alarmsHmi.message[#i].%X5 := #alarmsPlc.messages.msgNo[#x + 6];
       #alarmsHmi.message[#i].%X6 := #alarmsPlc.messages.msgNo[#x + 7];
       #alarmsHmi.message[#i].%X7 := #alarmsPlc.messages.msgNo[#x + 8];
       #alarmsHmi.message[#i].%X8 := #alarmsPlc.messages.msgNo[#x + 9];
       #alarmsHmi.message[#i].%X9 := #alarmsPlc.messages.msgNo[#x + 10];
       #alarmsHmi.message[#i].%X10 := #alarmsPlc.messages.msgNo[#x + 11];
       #alarmsHmi.message[#i].%X11 := #alarmsPlc.messages.msgNo[#x + 12];
       #alarmsHmi.message[#i].%X12 := #alarmsPlc.messages.msgNo[#x + 13];
       #alarmsHmi.message[#i].%X13 := #alarmsPlc.messages.msgNo[#x + 14];
       #alarmsHmi.message[#i].%X14 := #alarmsPlc.messages.msgNo[#x + 15];
       #alarmsHmi.message[#i].%X15 := #alarmsPlc.messages.msgNo[#x + 16];
   END_FOR;



   // set error 
   #error := false;
   FOR #i := 1 TO #lengthPlcErrors DO
       IF #alarmsPlc.alarms.errorNo[#i] THEN
           #error:= TRUE;
           EXIT;
       END_IF;
   END_FOR;


   // set message
   #message := false;
   FOR #i := 1 TO #lengthPlcMessages DO
       IF #alarmsPlc.messages.msgNo[#i] THEN
           #message := TRUE;
           EXIT;
       END_IF;
   END_FOR;
END_FUNCTION_BLOCK

// folder: 9. Library/9.1 Framework Functions

FUNCTION "SetError" : Void   // FC900, FBD
TITLE = Setze Fehler
{ S7_Optimized_Access := 'TRUE' }
VERSION : 0.1
// Ersteller: Andreas Fast Automation
// E-Mail: automation@fast-andreas.de
// 
// Projekt dient zu Demonstrationszwecken und frei genutzt werden.
// 
// Bausteinbeschreibung:
   VAR_INPUT
      trigger : Bool;   // Auslöser
      logic : Bool;   // Auslöserlogik; 0 = trigger ausgelöst bei false
   END_VAR
   VAR_OUTPUT
      error : Bool;
   END_VAR
BEGIN

REGION Network 1
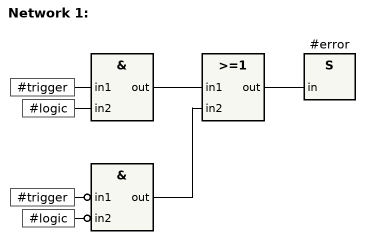
   IF (#trigger AND #logic) OR (NOT #trigger AND NOT #logic) THEN #error := TRUE; END_IF;
END_REGION
END_FUNCTION

FUNCTION "CheckAllStationsStopped" : Void   // FC901, SCL
{ S7_Optimized_Access := 'TRUE' }
VERSION : 0.1
   VAR_OUTPUT
      stopped : Bool;   // All stations are stopped
   END_VAR
   VAR_IN_OUT
      stations : "typeStations";
   END_VAR
   VAR_TEMP
      tempCounter : USInt;
   END_VAR
BEGIN
   // Ersteller: Andreas Fast Automation
   // E-Mail: automation@fast-andreas.de
   //
   // Projekt dient zu Demonstrationszwecken und frei genutzt werden.
   //
   // Bausteinbeschreibung:
   // 

   #stopped := true;

   FOR #tempCounter := 1 TO "SYS_MACHINE_MAXSTATIONS" DO
       // Check if all stations are stopped
       IF NOT #stations.station[#tempCounter].signals.isStopped AND #stations.station[#tempCounter].exists THEN
           #stopped := false;
           RETURN;
       END_IF;
   END_FOR;
END_FUNCTION

FUNCTION "CheckAnyStationError" : Void   // FC902, SCL
{ S7_Optimized_Access := 'TRUE' }
VERSION : 0.1
// Check if any station is in error
   VAR_OUTPUT
      error : Bool;
   END_VAR
   VAR_IN_OUT
      stations : "typeStations";
   END_VAR
   VAR_TEMP
      tempCounter : USInt;
   END_VAR
BEGIN
   // Ersteller: Andreas Fast Automation
   // E-Mail: automation@fast-andreas.de
   //
   // Projekt dient zu Demonstrationszwecken und frei genutzt werden.
   //
   // Bausteinbeschreibung:
   // 

   #error := false;

   FOR #tempCounter := 1 TO "SYS_MACHINE_MAXSTATIONS" DO
       // Check for error in stations
       IF #stations.station[#tempCounter].signals.isInError AND #stations.station[#tempCounter].exists THEN
           #error := true;
           RETURN;
       END_IF;
   END_FOR;
END_FUNCTION

FUNCTION "CheckAnyStationInSetup" : Void   // FC903, SCL
{ S7_Optimized_Access := 'TRUE' }
VERSION : 0.1
// Check if any station is in error
   VAR_OUTPUT
      setupActive : Bool;
   END_VAR
   VAR_IN_OUT
      stations : "typeStations";
   END_VAR
   VAR_TEMP
      tempCounter : USInt;
   END_VAR
BEGIN
   // Ersteller: Andreas Fast Automation
   // E-Mail: automation@fast-andreas.de
   //
   // Projekt dient zu Demonstrationszwecken und frei genutzt werden.
   //
   // Bausteinbeschreibung:
   // 

   #setupActive := false;

   FOR #tempCounter := 1 TO "SYS_MACHINE_MAXSTATIONS" DO
       // Check for error in stations
       IF #stations.station[#tempCounter].signals.setupActive AND #stations.station[#tempCounter].exists THEN
           #setupActive := true;
           RETURN;
       END_IF;
   END_FOR;
END_FUNCTION

FUNCTION "CheckAllStationsInHome" : Void   // FC904, SCL
{ S7_Optimized_Access := 'TRUE' }
VERSION : 0.1
   VAR_OUTPUT
      areInHome : Bool;   // All stations are in home
   END_VAR
   VAR_IN_OUT
      stations : "typeStations";
   END_VAR
   VAR_TEMP
      tempCounter : USInt;
   END_VAR
BEGIN
   // Ersteller: Andreas Fast Automation
   // E-Mail: automation@fast-andreas.de
   //
   // Projekt dient zu Demonstrationszwecken und frei genutzt werden.
   //
   // Bausteinbeschreibung:
   // 

   #areInHome := true;

   FOR #tempCounter := 1 TO "SYS_MACHINE_MAXSTATIONS" DO
       // Check if all stations are stopped
       IF NOT #stations.station[#tempCounter].signals.isInHome AND #stations.station[#tempCounter].exists THEN
           #areInHome := false;
           RETURN ;
       END_IF;
   END_FOR;
END_FUNCTION

FUNCTION "CheckAllStationsAutoRunning" : Void   // FC905, SCL
{ S7_Optimized_Access := 'TRUE' }
VERSION : 0.1
   VAR_OUTPUT
      running : Bool;   // All stations in automatic run
   END_VAR
   VAR_IN_OUT
      stations : "typeStations";
   END_VAR
   VAR_TEMP
      tempCounter : USInt;
   END_VAR
BEGIN
   // Ersteller: Andreas Fast Automation
   // E-Mail: automation@fast-andreas.de
   //
   // Projekt dient zu Demonstrationszwecken und frei genutzt werden.
   //
   // Bausteinbeschreibung:
   // 

   #running := true;

   FOR #tempCounter := 1 TO "SYS_MACHINE_MAXSTATIONS" DO
       // Check if all stations are stopped
       IF NOT #stations.station[#tempCounter].signals.releaseCycle
           AND #stations.station[#tempCounter].exists
       THEN
           #running := false;
           RETURN;
       END_IF;
   END_FOR;
END_FUNCTION

FUNCTION "CheckAnyStationInAutoRun" : Void   // FC906, SCL
{ S7_Optimized_Access := 'TRUE' }
VERSION : 0.1
   VAR_OUTPUT
      running : Bool;   // All stations in automatic run
   END_VAR
   VAR_IN_OUT
      stations : "typeStations";
   END_VAR
   VAR_TEMP
      tempCounter : USInt;
   END_VAR
BEGIN
   // Ersteller: Andreas Fast Automation
   // E-Mail: automation@fast-andreas.de
   //
   // Projekt dient zu Demonstrationszwecken und frei genutzt werden.
   //
   // Bausteinbeschreibung:
   // 

   #running := false;

   FOR #tempCounter := 1 TO "SYS_MACHINE_MAXSTATIONS" DO
       // Check if all stations are stopped
       IF //#stations.station[#tempCounter].signals.modeAuto AND
           #stations.station[#tempCounter].signals.releaseCycle
           AND #stations.station[#tempCounter].exists
       THEN
           #running := true;
           RETURN;
       END_IF;
   END_FOR;
END_FUNCTION

FUNCTION "S7GraphParameters" : Void   // FC910, FBD
TITLE = Steuerung Graph Parameter
{ S7_Optimized_Access := 'TRUE' }
VERSION : 0.1
// Ersteller: Andreas Fast Automation
// E-Mail: automation@fast-andreas.de
// 
// Projekt dient zu Demonstrationszwecken und frei genutzt werden.
// 
// Bausteinbeschreibung:
   VAR_OUTPUT
      ack : Bool;   // Schrittkette quittieren
      init : Bool;   // Schrittkette in Initialschritt schalten
      auto : Bool;   // Automatikbetrieb
      man : Bool;   // Handbetrieb
      tap : Bool;   // Halbautomatischer Betrieb
      push : Bool;   // Schaltfreigabe für Transition im halbautomatischen Betrieb
   END_VAR
   VAR_IN_OUT
      signals : "typeStationSignals";
   END_VAR
BEGIN

REGION Network 1: Schrittkette in Initialschritt schalten
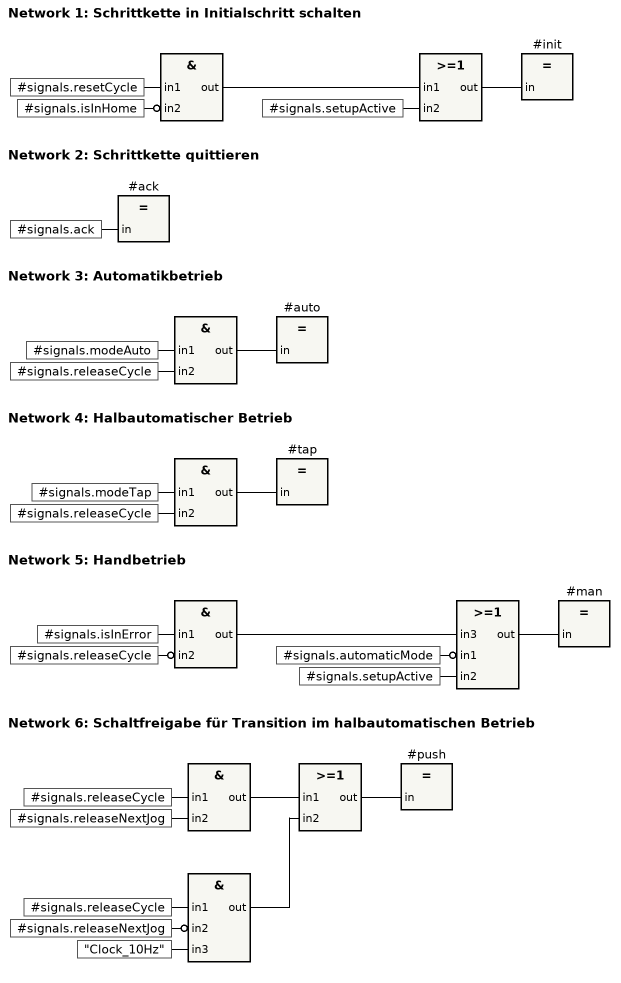
   #init := (#signals.resetCycle AND NOT #signals.isInHome) OR #signals.setupActive;
END_REGION

REGION Network 2: Schrittkette quittieren
   #ack := #signals.ack;
END_REGION

REGION Network 3: Automatikbetrieb
   #auto := #signals.modeAuto AND #signals.releaseCycle;
END_REGION

REGION Network 4: Halbautomatischer Betrieb
   #tap := #signals.modeTap AND #signals.releaseCycle;
END_REGION

REGION Network 5: Handbetrieb
   #man := (#signals.isInError AND NOT #signals.releaseCycle) OR NOT #signals.automaticMode OR #signals.setupActive;
END_REGION

REGION Network 6: Schaltfreigabe für Transition im halbautomatischen Betrieb
   #push := (#signals.releaseCycle AND #signals.releaseNextJog) OR (#signals.releaseCycle AND NOT #signals.releaseNextJog AND "Clock_10Hz");
END_REGION
END_FUNCTION

FUNCTION "CheckStepSeqError" : Void   // FC911, SCL
{ S7_Optimized_Access := 'TRUE' }
VERSION : 0.1
   VAR_OUTPUT
      error : Bool;
   END_VAR
   VAR_IN_OUT
      stepSequences : "typeStepSequences";
   END_VAR
   VAR_TEMP
      tempCounter : USInt;
   END_VAR
BEGIN
   // Ersteller: Andreas Fast Automation
   // E-Mail: automation@fast-andreas.de
   //
   // Projekt dient zu Demonstrationszwecken und frei genutzt werden.
   //
   // Bausteinbeschreibung:
   // 

   #error := false;



   FOR #tempCounter := 1 TO "SYS_SQ_MAXSEQUENCES" DO
       // Check for error in stations
       IF #stepSequences.stepSeq[#tempCounter].error AND #stepSequences.stepSeq[#tempCounter].exists THEN
           #error := true;
           RETURN;
       END_IF;
   END_FOR;
END_FUNCTION

FUNCTION "CheckStepSeqAllInHome" : Void   // FC912, SCL
{ S7_Optimized_Access := 'TRUE' }
VERSION : 0.1
   VAR_OUTPUT
      allInHome : Bool;   // Alle Schrittketten in Grundstellung
   END_VAR
   VAR_IN_OUT
      stepSequences : "typeStepSequences";
   END_VAR
   VAR_TEMP
      tempCounter : USInt;
   END_VAR
BEGIN
   // Ersteller: Andreas Fast Automation
   // E-Mail: automation@fast-andreas.de
   //
   // Projekt dient zu Demonstrationszwecken und frei genutzt werden.
   //
   // Bausteinbeschreibung:
   // 

   #allInHome := true;



   FOR #tempCounter := 1 TO "SYS_SQ_MAXSEQUENCES" DO
       // Check for error in stations
       IF NOT #stepSequences.stepSeq[#tempCounter].inHome AND #stepSequences.stepSeq[#tempCounter].exists THEN
           #allInHome := false;
           RETURN;
       END_IF;
   END_FOR;
END_FUNCTION

FUNCTION "CheckStepSeqAreWaiting" : Void   // FC913, SCL
{ S7_Optimized_Access := 'TRUE' }
VERSION : 0.1
   VAR_OUTPUT
      areWaiting : Bool;   // are waiting or in error
   END_VAR
   VAR_IN_OUT
      stepSequences : "typeStepSequences";
   END_VAR
   VAR_TEMP
      tempCounter : USInt;
   END_VAR
BEGIN
   // Ersteller: Andreas Fast Automation
   // E-Mail: automation@fast-andreas.de
   //
   // Projekt dient zu Demonstrationszwecken und frei genutzt werden.
   //
   // Bausteinbeschreibung:
   // 

   #areWaiting := true;


   FOR #tempCounter := 1 TO "SYS_SQ_MAXSEQUENCES" DO
       // Check for error in stations
       IF NOT #stepSequences.stepSeq[#tempCounter].isWaiting AND NOT #stepSequences.stepSeq[#tempCounter].error AND #stepSequences.stepSeq[#tempCounter].exists THEN
           #areWaiting := false;
           RETURN;
       END_IF;
   END_FOR;
END_FUNCTION

FUNCTION "CheckStepSeqAllJogDone" : Void   // FC914, SCL
{ S7_Optimized_Access := 'TRUE' }
VERSION : 0.1
   VAR_OUTPUT
      allJogDone : Bool;   // Alle Schrittketten haben halbautomatische Weiterschaltung abgeschlossen
   END_VAR
   VAR_IN_OUT
      signals : "typeStationSignals";
      stepSequences : "typeStepSequences";
   END_VAR
   VAR_TEMP
      tempCounter : USInt;
   END_VAR
BEGIN
   // Ersteller: Andreas Fast Automation
   // E-Mail: automation@fast-andreas.de
   //
   // Projekt dient zu Demonstrationszwecken und frei genutzt werden.
   //
   // Bausteinbeschreibung:
   // 

   #allJogDone := false;

   IF (#signals.modeTap AND NOT #signals.releaseNextJog) THEN // OR (#signals.modeAuto AND #signals.autoIsStoping) THEN

       #allJogDone := #signals.releaseCycle;

       FOR #tempCounter := 1 TO "SYS_SQ_MAXSEQUENCES" DO
           // Check if step sequence is done and exists
           IF NOT #stepSequences.stepSeq[#tempCounter].jogDone AND NOT #stepSequences.stepSeq[#tempCounter].isWaiting AND NOT #stepSequences.stepSeq[#tempCounter].error  AND #stepSequences.stepSeq[#tempCounter].exists THEN
               #allJogDone := false;
               RETURN;
           END_IF;
       END_FOR;
   ELSE
       #allJogDone := false;
   END_IF;
END_FUNCTION

FUNCTION "CheckAnyJogIsActive" : Void   // FC915, SCL
{ S7_Optimized_Access := 'TRUE' }
VERSION : 0.1
   VAR_OUTPUT
      anyJogIsActive : Bool;   // Mindestens eine Schrittketten läuft noch in halbautomatischer Weiterschaltung
   END_VAR
   VAR_IN_OUT
      stations : "typeStations";
   END_VAR
   VAR_TEMP
      tempCounter : USInt;
   END_VAR
BEGIN
   // Ersteller: Andreas Fast Automation
   // E-Mail: automation@fast-andreas.de
   //
   // Projekt dient zu Demonstrationszwecken und frei genutzt werden.
   //
   // Bausteinbeschreibung:
   // 

   #anyJogIsActive := false;

   FOR #tempCounter := 1 TO "SYS_MACHINE_MAXSTATIONS" DO

       IF #stations.station[#tempCounter].exists AND
           #stations.station[#tempCounter].signals.modeTap AND
           #stations.station[#tempCounter].signals.releaseCycle
       THEN
           #anyJogIsActive := true;
           RETURN;
       END_IF;

   END_FOR;
END_FUNCTION

FUNCTION "S7GraphInterlock" : Void   // FC919, FBD
TITLE = S7G Verriegelung (notwendig für den Einzelschritt)
{ S7_Optimized_Access := 'TRUE' }
VERSION : 0.1
// Ersteller: Andreas Fast Automation
// E-Mail: automation@fast-andreas.de
// 
// Projekt dient zu Demonstrationszwecken und frei genutzt werden.
// 
// Bausteinbeschreibung:
   VAR_INPUT
      interlock : Bool;   // Verriegelung
      setting : Bool;   // Verriegelungslogik (interlock == setting -> out wird freigegeben)
      alarm : Bool;   // Beim Alarm wird out rückgesetzt
   END_VAR
   VAR_OUTPUT
      out : Bool;
   END_VAR
BEGIN

REGION Network 1
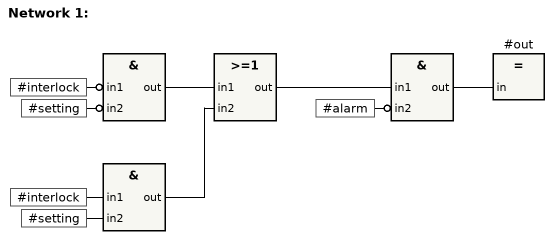
   #out := ((NOT #interlock AND NOT #setting) OR (#interlock AND #setting)) AND NOT #alarm;
END_REGION
END_FUNCTION

// folder: 9. Library/9.1 Framework Functions/ManualMovement

FUNCTION_BLOCK "ActorManualMovement"   // FB909, FBD
TITLE = Steuerung Einrichtbewegung eines Aktors
{ S7_Optimized_Access := 'TRUE' }
VERSION : 0.1
// Ersteller: Andreas Fast Automation
// E-Mail: automation@fast-andreas.de
// 
// Projekt dient zu Demonstrationszwecken und frei genutzt werden.
// 
// Bausteinbeschreibung:
   VAR_INPUT
      showValue : Bool;
      isExecutableRight : Bool;
      isExecutableLeft : Bool;
      showEndPositionRight : Bool;   // Sichtbarkeit rechte Seite
      showEndPositionLeft : Bool;   // Sichtbarkeit linke Seite
   END_VAR
   VAR_OUTPUT
      manualMoveNo : UInt;
   END_VAR
   VAR_IN_OUT
      manualWorkPos : Bool;   // Manueller Ansteuerbefehl für Arbeitsstellung
      manualHomePos : Bool;   // Manueller Ansteuerbefehl für Grundstellung
      actor : "typeActor";
      signals : "typeStationSignals";
      manualMovement : "typeManualMovements";
   END_VAR
   VAR
      statManualMovementNo : UInt;
      statStationNo : USInt;
      statMoveNoInStation : UInt;
   END_VAR
   VAR_TEMP
      tempInitialised : Bool;
      tempRelease : Bool;
   END_VAR
   VAR_TEMP   // added for the SCL form of the ladder/FBD networks
      _w1 : Bool;
   END_VAR
BEGIN

REGION Network 1: Initialisierungsprozess für eine Einrichtfunktion
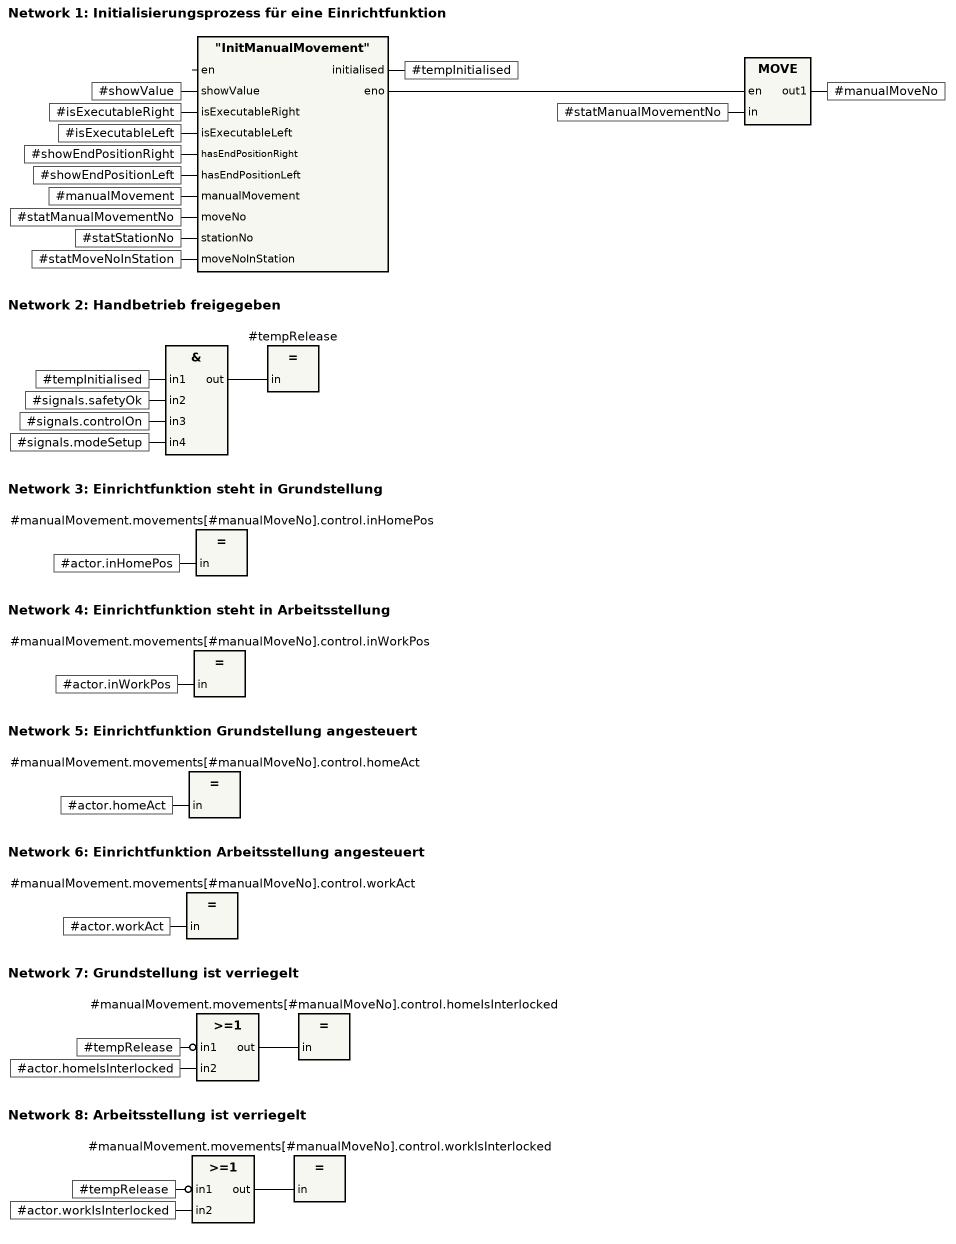
   "InitManualMovement"(showValue := #showValue,
                        isExecutableRight := #isExecutableRight,
                        isExecutableLeft := #isExecutableLeft,
                        hasEndPositionRight := #showEndPositionRight,
                        hasEndPositionLeft := #showEndPositionLeft,
                        manualMovement := #manualMovement,
                        moveNo := #statManualMovementNo,
                        stationNo := #statStationNo,
                        moveNoInStation := #statMoveNoInStation,
                        initialised => #tempInitialised,
                        ENO => #_w1);
   IF #_w1 THEN #manualMoveNo := #statManualMovementNo; END_IF;
END_REGION

REGION Network 2: Handbetrieb freigegeben
   #tempRelease := #tempInitialised AND #signals.safetyOk AND #signals.controlOn AND #signals.modeSetup;
END_REGION

REGION Network 3: Einrichtfunktion steht in Grundstellung
   #manualMovement.movements[#manualMoveNo].control.inHomePos := #actor.inHomePos;
END_REGION

REGION Network 4: Einrichtfunktion steht in Arbeitsstellung
   #manualMovement.movements[#manualMoveNo].control.inWorkPos := #actor.inWorkPos;
END_REGION

REGION Network 5: Einrichtfunktion Grundstellung angesteuert
   #manualMovement.movements[#manualMoveNo].control.homeAct := #actor.homeAct;
END_REGION

REGION Network 6: Einrichtfunktion Arbeitsstellung angesteuert
   #manualMovement.movements[#manualMoveNo].control.workAct := #actor.workAct;
END_REGION

REGION Network 7: Grundstellung ist verriegelt
   #manualMovement.movements[#manualMoveNo].control.homeIsInterlocked := NOT #tempRelease OR #actor.homeIsInterlocked;
END_REGION

REGION Network 8: Arbeitsstellung ist verriegelt
   #manualMovement.movements[#manualMoveNo].control.workIsInterlocked := NOT #tempRelease OR #actor.workIsInterlocked;
END_REGION

REGION Network 9: Rücksetze manuelle Bewegungsansteuerung des Aktors
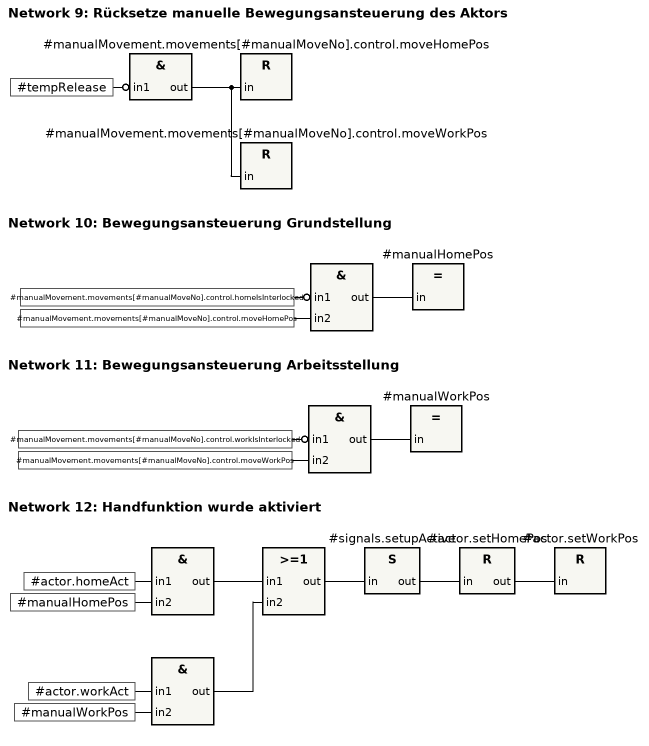
   IF NOT #tempRelease THEN
       #manualMovement.movements[#manualMoveNo].control.moveHomePos := FALSE;
       #manualMovement.movements[#manualMoveNo].control.moveWorkPos := FALSE;
   END_IF;
END_REGION

REGION Network 10: Bewegungsansteuerung Grundstellung
   #manualHomePos := NOT #manualMovement.movements[#manualMoveNo].control.homeIsInterlocked AND #manualMovement.movements[#manualMoveNo].control.moveHomePos;
END_REGION

REGION Network 11: Bewegungsansteuerung Arbeitsstellung
   #manualWorkPos := NOT #manualMovement.movements[#manualMoveNo].control.workIsInterlocked AND #manualMovement.movements[#manualMoveNo].control.moveWorkPos;
END_REGION

REGION Network 12: Handfunktion wurde aktiviert
   IF (#actor.homeAct AND #manualHomePos) OR (#actor.workAct AND #manualWorkPos) THEN
       #signals.setupActive := TRUE;
       #actor.setHomePos := FALSE;
       #actor.setWorkPos := FALSE;
   END_IF;
END_REGION
END_FUNCTION_BLOCK

FUNCTION_BLOCK "DriveManualMovementJog"   // FB910, FBD
TITLE = Einrichtfunktion Tippen für einen Servo
{ S7_Optimized_Access := 'TRUE' }
VERSION : 0.1
// Ersteller: Andreas Fast Automation
// E-Mail: automation@fast-andreas.de
// 
// Projekt dient zu Demonstrationszwecken und frei genutzt werden.
// 
// Bausteinbeschreibung:
   VAR_INPUT
      status : "typeDriveStatus";   // Status
   END_VAR
   VAR_OUTPUT
      manualMoveNo : UInt;
   END_VAR
   VAR_IN_OUT
      control : "typeDriveControl";   // Steuerbefehle
      signals : "typeStationSignals";
      manualMovement : "typeManualMovements";
   END_VAR
   VAR
      statActor : "typeActor";
      instActorManualMovement : "ActorManualMovement";
   END_VAR
   VAR_TEMP
      tempInitialised : Bool;
      tempRelease : Bool;
   END_VAR
BEGIN

REGION Network 1: steht in Grundstellung
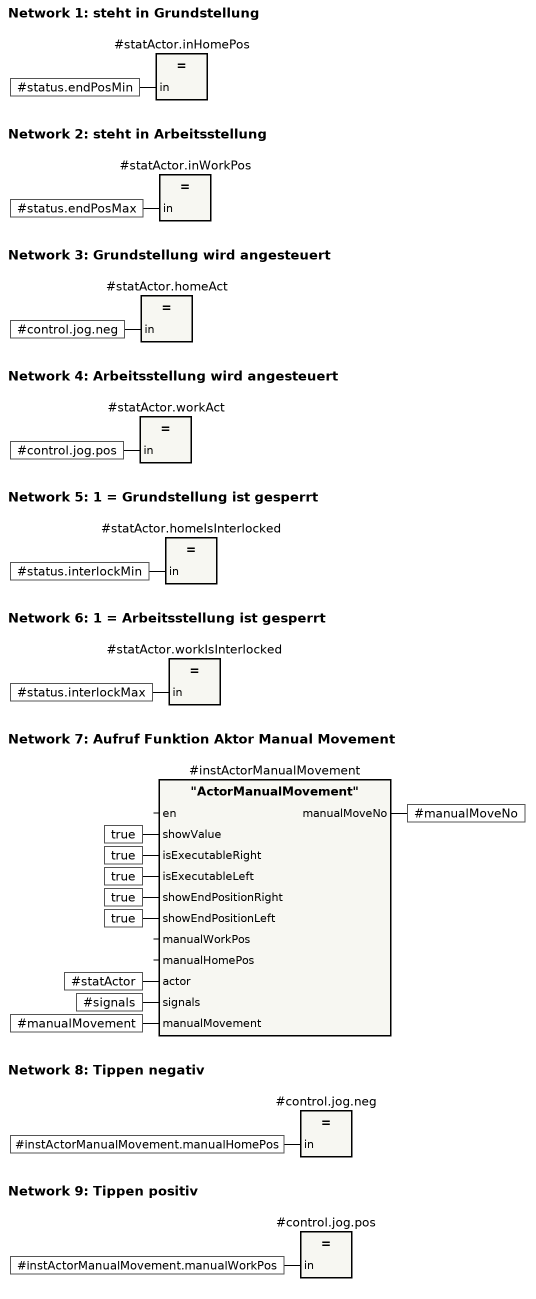
   #statActor.inHomePos := #status.endPosMin;
END_REGION

REGION Network 2: steht in Arbeitsstellung
   #statActor.inWorkPos := #status.endPosMax;
END_REGION

REGION Network 3: Grundstellung wird angesteuert
   #statActor.homeAct := #control.jog.neg;
END_REGION

REGION Network 4: Arbeitsstellung wird angesteuert
   #statActor.workAct := #control.jog.pos;
END_REGION

REGION Network 5: 1 = Grundstellung ist gesperrt
   #statActor.homeIsInterlocked := #status.interlockMin;
END_REGION

REGION Network 6: 1 = Arbeitsstellung ist gesperrt
   #statActor.workIsInterlocked := #status.interlockMax;
END_REGION

REGION Network 7: Aufruf Funktion Aktor Manual Movement
   #instActorManualMovement(showValue := true,   // "ActorManualMovement"
                           isExecutableRight := true,
                           isExecutableLeft := true,
                           showEndPositionRight := true,
                           showEndPositionLeft := true,
                           actor := #statActor,
                           signals := #signals,
                           manualMovement := #manualMovement,
                           manualMoveNo => #manualMoveNo);
END_REGION

REGION Network 8: Tippen negativ
   #control.jog.neg := #instActorManualMovement.manualHomePos;
END_REGION

REGION Network 9: Tippen positiv
   #control.jog.pos := #instActorManualMovement.manualWorkPos;
END_REGION

REGION Network 10: Istposition in Einrichtfunktion anzeigen
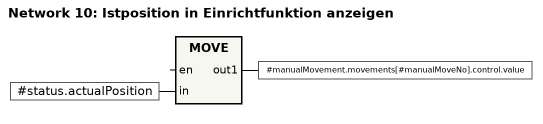
   #manualMovement.movements[#manualMoveNo].control.value := #status.actualPosition;
END_REGION
END_FUNCTION_BLOCK

FUNCTION "InitManualMovement" : Void   // FC907, FBD
TITLE = Initialisierungsprozess für eine Einrichtfunktion
{ S7_Optimized_Access := 'TRUE' }
VERSION : 0.1
// Ersteller: Andreas Fast Automation
// E-Mail: automation@fast-andreas.de
// 
// Projekt dient zu Demonstrationszwecken und frei genutzt werden.
// 
// Bausteinbeschreibung:
   VAR_INPUT
      showValue : Bool;   // Zeige Dezimalanzeige
      isExecutableRight : Bool;   // Ist ausführbar rechte Seite
      isExecutableLeft : Bool;   // Ist ausführbar linke Seite
      hasEndPositionRight : Bool;   // Zeige Endposition rechte Seite
      hasEndPositionLeft : Bool;   // Zeige Endposition linke Seite
   END_VAR
   VAR_OUTPUT
      initialised : Bool;
   END_VAR
   VAR_IN_OUT
      manualMovement : "typeManualMovements";
      moveNo : UInt;
      stationNo : USInt;
      moveNoInStation : UInt;
   END_VAR
   VAR_TEMP   // added for the SCL form of the ladder/FBD networks
      _w1 : Bool;
   END_VAR
BEGIN

REGION Network 1: Plausibilitätsprüfung/Initialisierung läuft
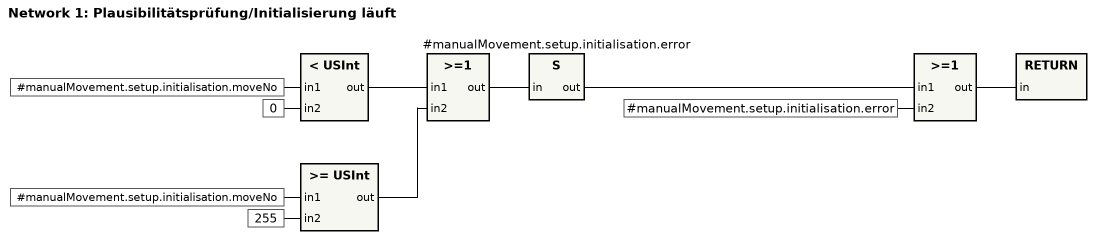
   #_w1 := (#manualMovement.setup.initialisation.moveNo < 0) OR (#manualMovement.setup.initialisation.moveNo >= 255);
   IF #_w1 THEN #manualMovement.setup.initialisation.error := TRUE; END_IF;
   IF #_w1 OR #manualMovement.setup.initialisation.error THEN
       ENO := TRUE;
       RETURN;
   END_IF;
END_REGION

REGION Network 2: Initialisierung
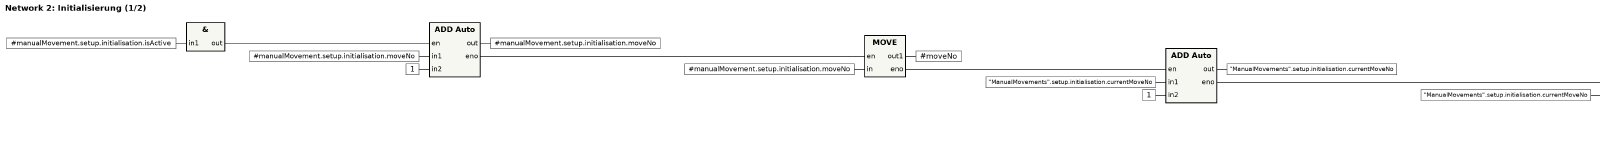
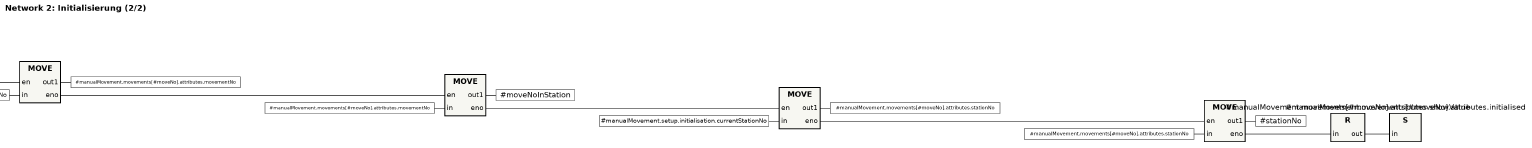
   IF #manualMovement.setup.initialisation.isActive THEN
       #manualMovement.setup.initialisation.moveNo := #manualMovement.setup.initialisation.moveNo + 1;
       #moveNo := #manualMovement.setup.initialisation.moveNo;
       "ManualMovements".setup.initialisation.currentMoveNo := "ManualMovements".setup.initialisation.currentMoveNo + 1;
       #manualMovement.movements[#moveNo].attributes.movementNo := "ManualMovements".setup.initialisation.currentMoveNo;
       #moveNoInStation := #manualMovement.movements[#moveNo].attributes.movementNo;
       #manualMovement.movements[#moveNo].attributes.stationNo := #manualMovement.setup.initialisation.currentStationNo;
       #stationNo := #manualMovement.movements[#moveNo].attributes.stationNo;
       #manualMovement.movements[#moveNo].attributes.showValue := FALSE;
       #manualMovement.movements[#moveNo].attributes.initialised := TRUE;
   END_IF;
END_REGION

REGION Network 3: Initialisierung abgeschlossen?
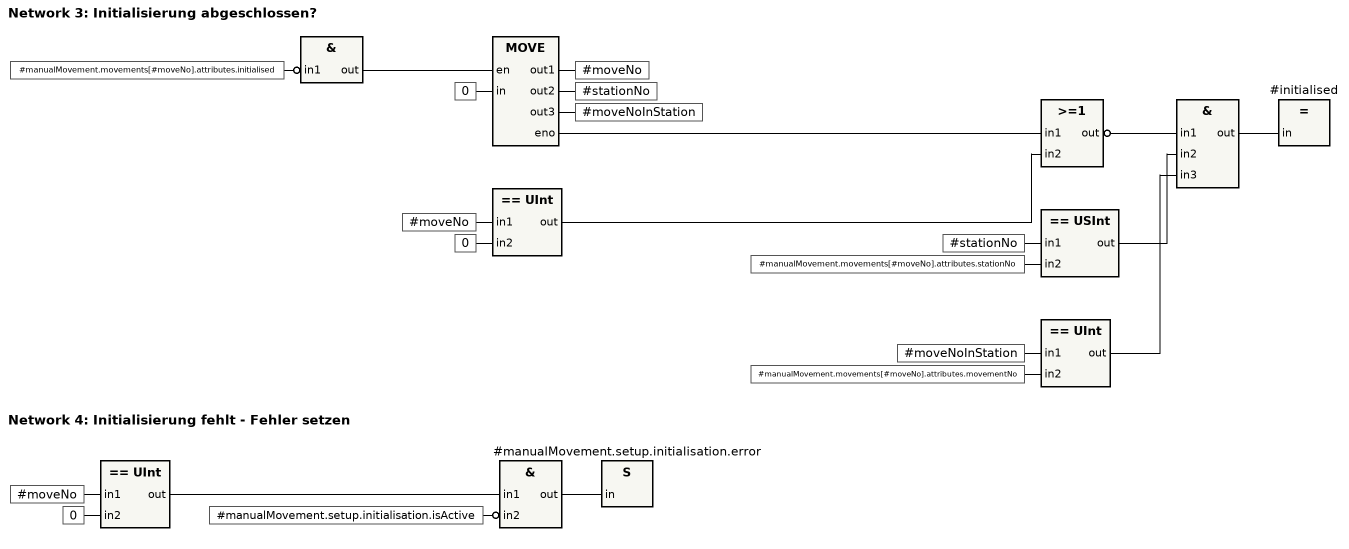
   #_w1 := NOT #manualMovement.movements[#moveNo].attributes.initialised;
   IF #_w1 THEN
       #moveNo := 0;
       #stationNo := 0;
       #moveNoInStation := 0;
   END_IF;
   #initialised := NOT (#_w1 OR (#moveNo = 0)) AND (#stationNo = #manualMovement.movements[#moveNo].attributes.stationNo) AND (#moveNoInStation = #manualMovement.movements[#moveNo].attributes.movementNo);
END_REGION

REGION Network 4: Initialisierung fehlt - Fehler setzen
   IF (#moveNo = 0) AND NOT #manualMovement.setup.initialisation.isActive THEN
       #manualMovement.setup.initialisation.error := TRUE;
   END_IF;
END_REGION

REGION Network 5: Sichtbarkeit
